// ---- GVLs/GlobalSettings.TcGVL
{attribute 'qualified_only'}
VAR_GLOBAL CONSTANT
	MAX_COMPONENTS: INT := 30;
	MAX_ALARMS: INT := 40;
END_VAR
{attribute 'qualified_only'}
VAR_GLOBAL PERSISTENT
	_dl:BOOL;
	{attribute 'TcEncoding':='UTF-8'}
	WebAdsAccessRoot: STRING := 'Main.GreenMaster';
	{attribute 'TcEncoding':='UTF-8'}
	PlcType: STRING := 'CX8190';
	PlcVersion: string := '1.0.33P5';
	Webname: STRING := 'NIBE AirSite GreenMaster';
	Users: ARRAY [0..24] OF User := [
		(Email := 'user', Password := 'user', Name := 'User', Permissions := Permissions.User),
		(Email := 'admin', Password := 'admin', Name := 'Admin', Permissions := Permissions.AdminUser),
		(Email := 'super', Password := 'super', Name := 'Super', Permissions := Permissions.SuperUser)
	];
	{attribute 'TcEncoding':='UTF-8'}
	SiteNames: ARRAY [0..99] OF STRING;
	Components: ARRAY [0..MAX_COMPONENTS - 1] OF Component := [
		(Name := ComponentNames.GM, EN := FALSE, Path := 'Main.GreenMaster', Required := TRUE, Permissions := Permissions.User),
		(Name := ComponentNames.GM_BASE, EN := TRUE, Path := 'Main.GreenMaster.Parameters', Required := TRUE, Resource := 'Parameter', Permissions := Permissions.User),
		(Name := ComponentNames.GM_IO, EN := TRUE, Path := 'Globals.IO', Required := TRUE, Resource := 'Parameter', Permissions := Permissions.User),
		(Name := ComponentNames.GM_VENT, EN := TRUE, Path := 'Main.GreenMaster.ParametersVENT', Resource := 'Parameter', Permissions := Permissions.User),
		(Name := ComponentNames.GM_XXL, EN := TRUE, Path := 'Main.GreenMaster.ParametersXXL', Resource := 'Parameter', Permissions := Permissions.User),
		(Name := ComponentNames.GM_A, EN := FALSE, Path := 'Main.GreenMaster.ParametersGMA', Resource := 'Parameter', Permissions := Permissions.User),
		(Name := ComponentNames.GM_C_F, EN := FALSE, Path := 'Main.GreenMaster.ParametersGMCF', Resource := 'Parameter', Permissions := Permissions.User),
		(Name := ComponentNames.GM_C_T, EN := FALSE, Path := 'Main.GreenMaster.ParametersGMCT', Resource := 'Parameter', Permissions := Permissions.User),
		(Name := ComponentNames.GM_SMOKE_CONTROL, EN := TRUE, Path := 'Main.GreenMaster.ParametersSC', Resource := 'Parameter', Permissions := Permissions.User),
		(Name := ComponentNames.SMOKE_CONTROL_ADS, EN := TRUE, Path := 'ADS_SmokeControl.Tags', Resource := 'Parameter', Permissions := Permissions.User),
		(Name := ComponentNames.GM_OPT_STD, EN := TRUE, Path := 'ADS_Standard.Tags', Resource := 'Parameter', Permissions := Permissions.User),
		(Name := ComponentNames.SIMULATION, EN := FALSE, Path := 'Main.GreenMaster.Simulation', Resource := 'Parameter', Permissions := Permissions.User),
		(Name := ComponentNames.REDUNDANCY, EN := FALSE, Path := 'Main.GreenMaster.Redundancy', Resource := 'Parameter', Permissions := Permissions.User),
		(Name := ComponentNames.EXTRA_ALARMS, EN := TRUE, Path := 'ADS_ExtraAlarms.Tags', Resource := 'Parameter', Permissions := Permissions.User),
		(Name := ComponentNames.PARALLEL_UNITS, EN := FALSE, Path := 'ADS_ParallelUnits.Tags', Resource := 'Parameter', Permissions := Permissions.User),
		(Name := ComponentNames.None)
	];
	AlarmDefs: ARRAY [0..MAX_ALARMS - 1] OF AlarmDef := [
		(Name := 'FireExtract', Polarity := AlarmPolarity.ActiveLow),
		(Name := '')
	];
END_VAR

// ---- POUs/Main.TcPOU
PROGRAM Main
VAR
	// JaWa
	_iDbg:INT;	
	_download5:BOOL;
	//Enum1: FanControlTypes := FanControlTypes.Flow;
	GreenMaster: GreenMasterXXL_FB;
	StartupDone: BOOL;
	EventLog: EventLog;
	xxx: bool;
	Saver: FB_S_UPS_CX81xx;
	HostName: FB_GetHostName;
	UseReverse_C_QN1: BOOL;
	test1: bool;
	
	Std_Interface : Standard_Interface;
	ExtraAlarms_Interface: ExtraAlarms_Interface;
	SmokeControl_Interface: SmokeControl_Interface;

	Redundancy:Redundancy;
	//ParallelUnits: ParallelUnits;
	
	GreenMasterDI: GreenMasterDI;
	GreenMasterDO: GreenMasterDO;
	GreenMasterAI: GreenMasterAI;
	GreenMasterAO: GreenMasterAO;
	GreenMasterAI2_RTU: GreenMasterAIU_ModbusRTU;
	AnySensorError: BOOL;
	{attribute 'TcEncoding':='UTF-8'}
	str: STRING;
	n: INT;
	
	DebugStop: BOOL;
	WritePersistentData: WritePersistentData;
	StartWritePersistentData: BOOL;
	SavedParameters: GreenMasterBaseParameters;
	DevMon: DeviationMonitor;
	DevValue: LREAL;
	TestPID: TestPID;
	fbTime : FB_LocalSystemTime := ( bEnable := TRUE, dwCycle := 1 );
	LastSecondsCounter: LINT;
    sTime: STRING;	
	sPart1: STRING;
	sPart2: STRING;
	ExceptionYet: BOOL;
	PTest: POINTER TO BYTE;
	Crash: BOOL;
	i: INT;
	w: WORD;
	Rr: LREAL;
	UseKL3464: BOOL;
	FreezeHysteresis: Hysteresis;
	CurrentFreezeAlarm: BOOL;
END_VAR
VAR PERSISTENT
END_VAR

IF NOT ExceptionYet THEN
	//__TRY
		EventLog(EventLogData := Globals.EventLog);
		IF NOT StartupDone THEN
			Globals.SystemStartTime := NowDT();
			EventLog.LogEvent(Message := 'Starting up', Kind := EventTypes.Information);
			//EventLog.LogEventJSON(Message := 'Test data $${KFactor} and $${PressureControl.SP}', Kind := EventTypes.Debug, VarAdr := ADR(GreenMaster.Parameters.Regulation.ExtractAir), VarSize := SIZEOF(GreenMaster.Parameters.Regulation.ExtractAir), VarType := 'AirParameters');
			Rr := 4;	
			i := -4;
			StartupDone := TRUE;
		END_IF
		SavedParameters := GreenMaster.GetParameters();
		Globals.SystemUpTime := DT_TO_DWORD(NowDT()) - DT_TO_DWORD(Globals.SystemStartTime);
		
		TestPID();
		
		str := '';
		FOR n := 0 TO GlobalSettings.MAX_COMPONENTS DO
			IF GlobalSettings.Components[n].Name = ComponentNames.NONE THEN
				EXIT;
			END_IF
			IF GlobalSettings.Components[n].EN THEN
				IF str <> '' THEN
					str := concat(str, ', ');
				END_IF
				str := concat(str, TO_STRING(GlobalSettings.Components[n].Name));
			END_IF
		END_FOR
		Globals.Components := str;
		
		HostName(bExecute := TRUE);
		// CX-503E98 CTH 1
		// CX-492F8F Diginet lab
		// CX-4F1CE6 NIBE AirSite lab
		// 
		Globals.HostName := HostName.sHostName; 
		IF F_ToUCase(HostName.sHostName) = 'CX-503E98' THEN
			UseReverse_C_QN1 := FALSE;
		ELSE
			UseReverse_C_QN1 := GreenMaster.Parameters.Io.AOutCalibration.C_QN1.InvertedOutput;
		END_IF
		
		IF F_ToUCase(HostName.sHostName) = 'STU_E6-LB02' THEN
			UseKL3464 := TRUE;
		END_IF
		IF (HostName.sHostName <> '') and (NOT GreenMaster.Parameters.System.ProjectDefaultSet) THEN			
			IF F_ToUCase(HostName.sHostName) = 'STU_E1-LB01' OR F_ToUCase(HostName.sHostName) = 'STU_E1-LB02' THEN
				GetComponent(Name := ComponentNames.PARALLEL_UNITS).EN := TRUE;
				GreenMaster.GetParameters().Regulation.Temperature.HeaterOutputDirection := HeaterOutputDirections.IncreaseToHeat;
				GreenMaster.GetParameters().Regulation.ExtractAir.Control.I := T#10M;
				GreenMaster.GetParameters().Regulation.SupplyAir.Control.I := T#10M;
				ADS_Standard.Tags.Settings.ExtractFanControl_I := GreenMaster.GetParameters().Regulation.ExtractAir.Control.I;
				ADS_Standard.Tags.Settings.SupplyFanControl_I := GreenMaster.GetParameters().Regulation.SupplyAir.Control.I;
				GreenMaster.GetParameters().Regulation.ExtractAir.KFactor := 151.4;
				GreenMaster.GetParameters().Regulation.ExtractAir.FireExhaust.EN := TRUE;
				GreenMaster.GetParameters().Regulation.ExtractAir.FireExhaust.Speed := 0.4;
				GreenMaster.GetParameters().Regulation.ExtractAir.FireSupply.EN := TRUE;
				GreenMaster.GetParameters().Regulation.ExtractAir.FireSupply.Speed := 0.4;
				GreenMaster.GetParameters().Regulation.SupplyAir.KFactor := 151.4;
				GreenMaster.GetParameters().Regulation.SupplyAir.FireExhaust.EN := FALSE;
				GreenMaster.GetParameters().Regulation.SupplyAir.FireExhaust.Speed := 0;
				GreenMaster.GetParameters().Alarm.Polarity.B.Tx1Fail := TRUE;
				GreenMaster.GetParameters().Alarm.Enabled.B.Pump1 := FALSE;
				ADS_ParallelUnits.Tags.Settings.SupplyAirSetPointAdjustment.Curve.Y1 := 160;
				ADS_ParallelUnits.Tags.Settings.SupplyAirSetPointAdjustment.Curve.Y2 := 160;
				ADS_ParallelUnits.Tags.Settings.SupplyAirSetPointAdjustment.Curve.Y3 := 160;
				ADS_ParallelUnits.Tags.Settings.SupplyAirSetPointAdjustment.Curve.Y4 := 160;
				ADS_ParallelUnits.Tags.Settings.SupplyAirSetPointAdjustment.Curve.Y5 := 160;
				ADS_ParallelUnits.Tags.Settings.SupplyAirSetPointAdjustment.Curve.Y6 := 160;
				ADS_ParallelUnits.Tags.Settings.SupplyAirSetPointAdjustment.Curve.Y7 := 160;
				ADS_ParallelUnits.Tags.Settings.SupplyAirSetPointAdjustment.Curve.Y8 := 160;
				ADS_ParallelUnits.Tags.Settings.SupplyAirSetPointAdjustment.Curve.Y9 := 160;
				
				ADS_ParallelUnits.Tags.Settings.ExtractAirSetPointAdjustment.Curve.Y1 := 150;
				ADS_ParallelUnits.Tags.Settings.ExtractAirSetPointAdjustment.Curve.Y2 := 150;
				ADS_ParallelUnits.Tags.Settings.ExtractAirSetPointAdjustment.Curve.Y3 := 150;
				ADS_ParallelUnits.Tags.Settings.ExtractAirSetPointAdjustment.Curve.Y4 := 150;
				ADS_ParallelUnits.Tags.Settings.ExtractAirSetPointAdjustment.Curve.Y5 := 150;
				ADS_ParallelUnits.Tags.Settings.ExtractAirSetPointAdjustment.Curve.Y6 := 150;
				ADS_ParallelUnits.Tags.Settings.ExtractAirSetPointAdjustment.Curve.Y7 := 150;
				ADS_ParallelUnits.Tags.Settings.ExtractAirSetPointAdjustment.Curve.Y8 := 150;
				ADS_ParallelUnits.Tags.Settings.ExtractAirSetPointAdjustment.Curve.Y9 := 150;
			END_IF
			IF F_ToUCase(HostName.sHostName) = 'STU_E6-LB03' THEN
				GreenMaster.GetParameters().Regulation.Temperature.HeaterOutputDirection := HeaterOutputDirections.DecreaseToHeat;
				GreenMaster.GetParameters().Regulation.ExtractAir.KFactor := 111;
				GreenMaster.GetParameters().Regulation.ExtractAir.FireExhaust.EN := FALSE;
				GreenMaster.GetParameters().Regulation.ExtractAir.FireExhaust.Speed := 0;
				GreenMaster.GetParameters().Regulation.ExtractAir.FireSupply.EN := FALSE;
				GreenMaster.GetParameters().Regulation.ExtractAir.FireSupply.Speed := 0;
				GreenMaster.GetParameters().Regulation.SupplyAir.KFactor := 111;
				GreenMaster.GetParameters().Regulation.SupplyAir.FireExhaust.EN := FALSE;
				GreenMaster.GetParameters().Regulation.SupplyAir.FireExhaust.Speed := 0;
				GreenMaster.GetParameters().Alarm.Polarity.B.Pump1 := TRUE;
			END_IF
			IF F_ToUCase(HostName.sHostName) = 'STU_E6-LB01' OR F_ToUCase(HostName.sHostName) = 'STU_E6-LB02' THEN
				GetComponent(Name := ComponentNames.PARALLEL_UNITS).EN := TRUE;
				GreenMaster.GetParameters().Regulation.Temperature.HeaterOutputDirection := HeaterOutputDirections.IncreaseToHeat;
				GreenMaster.GetParameters().Regulation.ExtractAir.KFactor := 111;
				GreenMaster.GetParameters().Regulation.ExtractAir.FireExhaust.EN := FALSE;
				GreenMaster.GetParameters().Regulation.ExtractAir.FireExhaust.Speed := 0;
				GreenMaster.GetParameters().Regulation.SupplyAir.KFactor := 111;
				GreenMaster.GetParameters().Regulation.SupplyAir.FireExhaust.EN := FALSE;
				GreenMaster.GetParameters().Regulation.SupplyAir.FireExhaust.Speed := 0;
				GreenMaster.GetParameters().Alarm.Polarity.B.Tx1Fail := TRUE;
			END_IF
			IF F_ToUCase(HostName.sHostName) = 'AIRPLC-DEMO' THEN
				GetComponent(Name := ComponentNames.PARALLEL_UNITS).EN := TRUE;
				GetComponent(Name := ComponentNames.SIMULATION).EN := TRUE;
				GreenMaster.GetParameters().System.Operation.Simulation := TRUE;
				GreenMaster.GetParameters().Regulation.Temperature.HeaterOutputDirection := HeaterOutputDirections.IncreaseToHeat;
				GreenMaster.GetParameters().Regulation.ExtractAir.KFactor := 111;
				GreenMaster.GetParameters().Regulation.ExtractAir.FireExhaust.EN := FALSE;
				GreenMaster.GetParameters().Regulation.ExtractAir.FireExhaust.Speed := 0;
				GreenMaster.GetParameters().Regulation.SupplyAir.KFactor := 111;
				GreenMaster.GetParameters().Regulation.SupplyAir.FireExhaust.EN := FALSE;
				GreenMaster.GetParameters().Regulation.SupplyAir.FireExhaust.Speed := 0;
				//GreenMaster.GetParameters().Regulation.SupplyAir.MaxSpeed := 0.4;
				//GreenMaster.GetParameters().Regulation.ExtractAir.MaxSpeed := 0.4;
			END_IF
			IF F_ToUCase(HostName.sHostName) = 'CX-662AA1' THEN
				GetComponent(Name := ComponentNames.PARALLEL_UNITS).EN := TRUE;
				GetComponent(Name := ComponentNames.SIMULATION).EN := TRUE;
				GreenMaster.GetParameters().System.Operation.Simulation := TRUE;
				GreenMaster.GetParameters().Regulation.Temperature.HeaterOutputDirection := HeaterOutputDirections.IncreaseToHeat;
				GreenMaster.GetParameters().Regulation.ExtractAir.KFactor := 111;
				GreenMaster.GetParameters().Regulation.ExtractAir.FireExhaust.EN := FALSE;
				GreenMaster.GetParameters().Regulation.ExtractAir.FireExhaust.Speed := 0;
				GreenMaster.GetParameters().Regulation.SupplyAir.KFactor := 111;
				GreenMaster.GetParameters().Regulation.SupplyAir.FireExhaust.EN := FALSE;
				GreenMaster.GetParameters().Regulation.SupplyAir.FireExhaust.Speed := 0;
				GreenMaster.GetParameters().Regulation.SupplyAir.MaxSpeed := 0.4;
				GreenMaster.GetParameters().Regulation.ExtractAir.MaxSpeed := 0.4;
			END_IF
			IF (F_ToUCase(HostName.sHostName) = 'DIGINET-1') or (F_ToUCase(HostName.sHostName) = 'DIGINET-2') THEN
				GetComponent(Name := ComponentNames.PARALLEL_UNITS).EN := TRUE;
				GetComponent(Name := ComponentNames.SIMULATION).EN := TRUE;
				GreenMaster.GetParameters().System.Operation.Simulation := TRUE;
				GreenMaster.GetParameters().Regulation.Temperature.HeaterOutputDirection := HeaterOutputDirections.IncreaseToHeat;
				GreenMaster.GetParameters().Regulation.ExtractAir.KFactor := 111;
				GreenMaster.GetParameters().Regulation.ExtractAir.FireExhaust.EN := TRUE;
				GreenMaster.GetParameters().Regulation.ExtractAir.FireExhaust.Speed := 0.5;
				GreenMaster.GetParameters().Regulation.SupplyAir.KFactor := 111;
				GreenMaster.GetParameters().Regulation.SupplyAir.FireExhaust.EN := FALSE;
				GreenMaster.GetParameters().Regulation.SupplyAir.FireExhaust.Speed := 0;
				GreenMaster.GetParameters().system.Operation.StartupHeatRecoveryTime := T#30S;
				GreenMaster.GetParameters().system.Operation.ExhaustFanStartupDelay := T#10S;
				GreenMaster.GetParameters().system.Operation.SupplyFanStartupDelay := T#20S;
				GreenMaster.GetParameters().system.Operation.StartupDamperWaitTime := T#5S;
			END_IF
			GreenMaster.GetParameters().System.ProjectDefaultSet := TRUE;
		END_IF
		
		IF GreenMaster.Parameters.System.Operation.IoUpdateEN THEN
			GreenMasterDI(DIn := Globals.IO.DIn, DInLevels := GreenMaster.Parameters.IO.DInLevels);
			GreenMasterDO(DOut := Globals.IO.DOut);
			GreenMasterAI(AIn := Globals.IO.AIn);
			GreenMasterAO(AOut := Globals.IO.AOut);
			GreenMasterAI2_RTU(Parameters:=GreenMaster.GetParameters(), EN:= TRUE);
		END_IF
		
		Std_Interface(EN := GetComponent(Name := ComponentNames.GM_OPT_STD).EN, AIn := Globals.IO.AIn);
		
		// Redundant drift
		IF GetComponent(Name := ComponentNames.REDUNDANCY).EN THEN
			Redundancy(	EN := GetComponent(Name := ComponentNames.REDUNDANCY).EN,
						_UPPSTART_DONE:=StartupDone,
						_TF_CMD:=GreenMaster.Parameters.Regulation.SupplyAir.Control.CV > 0,
						_TF_V:=GreenMaster.Parameters.Regulation.SupplyAir.Control.CV > 0 AND GreenMaster.GetCurrentSupplyAirPV() > 10,
						_TF_OP:=LREAL_TO_REAL(GreenMaster.Parameters.Regulation.SupplyAir.Control.CV),
						_TL_GP_PV:=LREAL_TO_REAL(GreenMaster.GetCurrentSupplyAirPV()),
						_FF_CMD:=GreenMaster.Parameters.Regulation.ExtractAir.Control.CV > 0,
						_FF_V:=GreenMaster.Parameters.Regulation.ExtractAir.Control.CV > 0 AND GreenMaster.GetCurrentExtractAirPV() > 10,
						_FF_OP:=LREAL_TO_REAL(GreenMaster.Parameters.Regulation.ExtractAir.Control.CV),
						_FL_GP_PV:=LREAL_TO_REAL(GreenMaster.GetCurrentExtractAirPV()),
						_SERVICEBRYTARE:=FALSE
						);
		END_IF
		// Parallel units
		(*
		IF GetComponent(Name := ComponentNames.PARALLEL_UNITS).EN THEN
			ParallelUnits(	EN := GetComponent(Name := ComponentNames.PARALLEL_UNITS).EN,
							Tags := ADS_ParallelUnits.Tags,
							Parameters := GreenMaster.Parameters 
						);
		END_IF
		*)
		IF GetComponent(Name := ComponentNames.GM_BASE).EN THEN
			GreenMaster.Update(DO_ := GreenMasterDO, AO := GreenMasterAO);
			GreenMaster(
				EN := TRUE AND (NOT DebugStop),
				RemoteEN := GreenMaster.Parameters.System.Operation.RemoteEN, //Std_Interface.ENO OR CTH_Interface.ENO OR Stena_Interface.ENO,	// TODO: Varför bara CTH här i original?  
				DI := GreenMasterDI,
				AI := GreenMasterAI,
				AI2 := GreenMasterAI2_RTU,
				TCP_AI := SmokeControl.GreenMasterSmokeControl,  
				Reverse_C_QN1 := UseReverse_C_QN1,
				NightCooling := GreenMaster.Parameters.Regulation.NightCooling,
				EnableFansAndDampers := Std_Interface.EN,
				ExtraFireSupplyAlarm := FALSE, //ParallelUnits.FireSupplyAlarm,
				ExtraFireExtractAlarm := FALSE //ParallelUnits.FireExtractAlarm
			);
		END_IF
		
		IF GetComponent(Name := ComponentNames.SIMULATION).EN THEN
			IF GreenMaster.GetParameters().System.Operation.Simulation THEN
				GreenMaster.Simulation(Parameters := GreenMaster.GetParameters(), Simulation := GreenMaster.GetParameters().Simulation);			
			END_IF
		END_IF
		
		AnySensorError := GreenMaster.Parameters.IO.AIn.F_BT1_Error OR 
			GreenMaster.Parameters.IO.AIn.T_BT2_Error OR
			GreenMaster.Parameters.IO.AIn.T_BT3_Error OR
			GreenMaster.Parameters.IO.AIn.H_BT1_Error OR
			GreenMaster.Parameters.IO.AIn.T_BT1_Error OR
			GreenMaster.Parameters.IO.AIn.BT1_Error OR
			GreenMaster.Parameters.IO.AIn.BT2_Error OR
			GreenMaster.Parameters.IO.AIn.F_BT2_Error OR	
			GreenMaster.Parameters.IO.AIn.F_BP1_Error OR
			GreenMaster.Parameters.IO.AIn.T_BP1_Error OR
			GreenMaster.Parameters.IO.AIn.F_BP2_Error OR
			GreenMaster.Parameters.IO.AIn.T_BP2_Error OR
			GreenMaster.Parameters.IO.AIn.F_BP3_Error OR
			GreenMaster.Parameters.IO.AIn.T_BF1_Error OR
			GreenMaster.Parameters.IO.AIn.F_BF1_Error;	
		
		
		// Save persistent data on power off or fail
		Saver();
		WritePersistentData(NETID := '', PORT := 851, TMOUT := T#10S, START := StartWritePersistentData);
		
		DevMon(Value := DevValue, TargetValue := 5);
		
		IF GetComponent(Name := ComponentNames.EXTRA_ALARMS).EN THEN	
			GreenMaster.GetParameters().Alarm.Status.A.AL01 := NOT ExtraAlarmInputs.AL01;
			GreenMaster.GetParameters().Alarm.Status.A.AL02 := NOT ExtraAlarmInputs.AL02;
			GreenMaster.GetParameters().Alarm.Status.A.AL03 := NOT ExtraAlarmInputs.AL03;
			GreenMaster.GetParameters().Alarm.Status.A.AL04 := NOT ExtraAlarmInputs.AL04;
			GreenMaster.GetParameters().Alarm.Status.A.AL05 := NOT ExtraAlarmInputs.AL05;
			GreenMaster.GetParameters().Alarm.Status.A.AL06 := NOT ExtraAlarmInputs.AL06;
			GreenMaster.GetParameters().Alarm.Status.A.AL07 := NOT ExtraAlarmInputs.AL07;
			GreenMaster.GetParameters().Alarm.Status.A.AL08 := NOT ExtraAlarmInputs.AL08;
		END_IF
		ExtraAlarms_Interface(EN := GetComponent(Name := ComponentNames.EXTRA_ALARMS).EN);
		SmokeControl_Interface(EN := GetComponent(Name := ComponentNames.GM_SMOKE_CONTROL).EN);
		fbtime();
		IF Globals.SecondsCounter <> LastSecondsCounter THEN
			LastSecondsCounter := Globals.SecondsCounter;
			// 2021-11-10-08:08:53.582
			sTime := SYSTEMTIME_TO_STRING(fbTime.systemTime);
			sPart1 := Delete(sTime, 4, 20);
			sPart2 := Replace(sPart1, ' ', 1, 11);
			GreenMaster.GetParameters().System.SystemTime := sPart2;
		END_IF
	//__CATCH
	//	ExceptionYet := TRUE; 			
	//__ENDTRY
ELSE
	ExceptionYet := TRUE; 	
END_IF

FreezeHysteresis(Value := GreenMaster.GetParameters().IO.AIn.H_BT1, LimitValue := GreenMaster.GetParameters().Alarm.Limits.A.Freeze, Offset := 0.5);
CurrentFreezeAlarm := FreezeHysteresis.Below OR GreenMaster.GetParameters().IO.AIn.H_BT1_Error;
GreenMaster.GetParameters().Alarm.Status.A.Freeze := CurrentFreezeAlarm  (*OR	ParallelUnits.FreezeAlarm*);

END_PROGRAM

// ---- POUs/GreenMasterXXL_FB.TcPOU
FUNCTION_BLOCK GreenMasterXXL_FB EXTENDS GreenMasterXXL
VAR_INPUT
END_VAR
VAR_OUTPUT
END_VAR
VAR
END_VAR


// PAGE Overview
Super^(); // GreenMasterXXL

END_FUNCTION_BLOCK

// ---- DUTs/GreenMaster/GreenMasterXXL.TcPOU
FUNCTION_BLOCK GreenMasterXXL EXTENDS GreenMasterBase
VAR
	ParametersXXLFB: GreenMasterParametersXXLFB;
END_VAR
VAR PERSISTENT
	ParametersXXL: GreenMasterParametersXXL;
END_VAR
VAR_INPUT
END_VAR
VAR_OUTPUT
END_VAR
VAR
	SupplyFanControl: FanControl;
	ExtractFanControl: FanControl;
	Recirculation: BOOL;
	VentilationControl: VentilationControl;
	ExhaustAir: BOOL;
	SupplyAir: BOOL := TRUE;
	StopVentilation: bool;

	ExtractFanPV: LREAL;
	SupplyFanPV: LREAL;
	Defrost_0: Defrost;
	WriteLRealIf_0: WriteLRealIf;
END_VAR
VAR // added by the converter: edge detectors and wires of the graphical bodies
    _w1, _w2, _w3, _w4 : ANY;
END_VAR


// PAGE Base functionality Inherited from greenMasterBase
Super^(); // GreenMasterBase

// PAGE Ventilation
Ventilation := VentilationControl.ENO;
VentilationControl(EN := Parameters.Regulation.Control.EN AND SystemStateVentilation AND ENO AND NOT StopVentilation);
VentilationRunning := VentilationControl.ENO;

// PAGE Supply Air
Parameters.Regulation.SupplyAir.Control.CV := SupplyFanControl.CV;
_w1 := Parameters.Alarm.Active.B.SupplyFan OR Parameters.Alarm.Active.B.ExtractFan;
WriteLRealIf_0(Out := Parameters.IO.AOut.T_GQ1, EN := TRUE, In := SupplyFanControl.CV); // WriteLRealIf
// Output via VAR_IN_OUT
SupplyFanControl(
    Parameters := Parameters,
    EN := Ventilation,
    ControlMode := Parameters.Regulation.SupplyAir.ControlMode,
    ControlParameters := Parameters.Regulation.SupplyAir.Control,
    Pressure := Parameters.IO.AIn.T_BP1,
    PressureError := Parameters.IO.Status.SensorStatus.T_BP1 <> 'OK',
    Flow := Parameters.IO.AIn.T_BF1,
    FlowError := Parameters.IO.Status.SensorStatus.T_BF1 <> 'OK',
    MasterPV := ExtractFanPV,
    FanAlarm := _w1,
    MinSpeed := Parameters.Regulation.SupplyAir.MinSpeed,
    MaxSpeed := Parameters.Regulation.SupplyAir.MaxSpeed,
    ExtendedOperation := _w2,
    PostVentilationTime := Parameters.System.Operation.PostVentilationTime,
    FireExhaust := GetFireExtractAlarms(),
    Damper := Parameters.IO.DOut.T_QM2,
    FireExhaustPar := Parameters.Regulation.SupplyAir.FireExhaust,
    FireSupplyPar := Parameters.Regulation.SupplyAir.FireSupply,
    FireSupply := Parameters.Alarm.Active.A.FireSupply); // FanControl
SupplyFanPV := SupplyFanControl.PV;
Parameters.IO.DOut.T_RUN := SupplyFanControl.FanRunning;
Parameters.IO.DOut.R_QM1 := SupplyFanControl.Recirculation;
_w2 := NightCooling OR DI.ExtendedOperation OR Parameters.System.Operation.TimeChannels.HighSpeed;

// PAGE Extract Air
_w3 := NightCooling OR DI.ExtendedOperation OR Parameters.System.Operation.TimeChannels.HighSpeed;
Parameters.Regulation.ExtractAir.Control.CV := ExtractFanControl.CV;
_w4 := Parameters.Alarm.Active.B.SupplyFan OR Parameters.Alarm.Active.B.ExtractFan;
WriteLRealIf_0(Out := Parameters.IO.AOut.F_GQ1, EN := TRUE, In := ExtractFanControl.CV); // WriteLRealIf
// Output via VAR_IN_OUT
ExtractFanControl(
    Parameters := Parameters,
    EN := Ventilation,
    ControlMode := Parameters.Regulation.ExtractAir.ControlMode,
    ControlParameters := Parameters.Regulation.ExtractAir.Control,
    Pressure := Parameters.IO.AIn.F_BP1,
    PressureError := Parameters.IO.Status.SensorStatus.F_BP1 <> 'OK',
    Flow := Parameters.IO.AIn.F_BF1,
    FlowError := Parameters.IO.Status.SensorStatus.F_BF1 <> 'OK',
    MasterPV := SupplyFanPV,
    FanAlarm := _w4,
    MinSpeed := Parameters.Regulation.ExtractAir.MinSpeed,
    MaxSpeed := Parameters.Regulation.ExtractAir.MaxSpeed,
    ExtendedOperation := _w3,
    PostVentilationTime := Parameters.System.Operation.PostVentilationTime,
    FireExhaust := GetFireExtractAlarms(),
    Damper := Parameters.IO.DOut.F_QM1,
    FireExhaustPar := Parameters.Regulation.ExtractAir.FireExhaust,
    FireSupplyPar := Parameters.Regulation.ExtractAir.FireSupply,
    FireSupply := Parameters.Alarm.Active.A.FireSupply); // FanControl
ExtractFanPV := ExtractFanControl.PV;
Parameters.IO.DOut.F_RUN := ExtractFanControl.FanRunning;

// PAGE Defrost
Defrost_0(
    Parameters := Parameters,
    EN := Parameters.System.Defrost.EN AND NOT Parameters.Alarm.Active.A.FireSupply AND NOT (GetFireExtractAlarms()),
    Temperature := Parameters.IO.AIn.T_BT2,
    Pressure := Parameters.IO.AIn.F_BP3); // Defrost

METHOD ExtractFanOverride : BOOL
VAR_INPUT
	Override: BOOL;
	Speed: LREAL;
END_VAR
VAR_INST
	LastExtractOverrideCV: lreal;
END_VAR
ExtractFanControl.Override := Override;
ExtractFanControl.OverrideCV := Speed;
ExtractFanControl.SyncCV := LastExtractOverrideCV;
IF Speed > 0 THEN
	LastExtractOverrideCV := Speed;
END_IF
END_METHOD

METHOD Fire : BOOL
VAR_INPUT
END_VAR
SUPER^.Fire();
SupplyFanControl.Override := Parameters.Regulation.SupplyAir.FireExhaust.EN;
SupplyFanControl.OverrideCV := Parameters.Regulation.SupplyAir.FireExhaust.Speed;
ExtractFanControl.Override := Parameters.Regulation.ExtractAir.FireExhaust.EN;
ExtractFanControl.OverrideCV := Parameters.Regulation.ExtractAir.FireExhaust.Speed;
END_METHOD

METHOD FireEnd : BOOL
VAR_INPUT
END_VAR
SUPER^.FireEnd();
SupplyFanControl.Override := FALSE;
SupplyFanControl.OverrideCV := 0;
ExtractFanControl.Override := FALSE;
ExtractFanControl.OverrideCV := 0;
END_METHOD

METHOD FireSupply : BOOL
VAR_INPUT
END_VAR
SUPER^.FireSupply();
CloseDampers();
StopVentilation := TRUE;
END_METHOD

METHOD FireSupplyEnd : BOOL
VAR_INPUT
END_VAR
SUPER^.FireSupplyEnd();
StopVentilation := FALSE;
END_METHOD

METHOD GetParametersXXL : REFERENCE TO GreenMasterParametersXXL
VAR_INPUT
END_VAR
GetParametersXXL := ParametersXXL;
END_METHOD

{attribute 'TcRpcEnable'}
METHOD Sum : LREAL
VAR_INPUT
	v1: LREAL;
	v2: LREAL;
END_VAR
Sum := v1 + v2;
END_METHOD

METHOD SupplyFanOverride : BOOL
VAR_INPUT
	Override: BOOL;
	Speed: LREAL;
END_VAR
VAR_INST
	LastSupplyOverrideCV: lreal;
END_VAR
SupplyFanControl.Override := Override;
SupplyFanControl.OverrideCV := Speed;
SupplyFanControl.SyncCV := LastSupplyOverrideCV;
IF Speed > 0 THEN
	LastSupplyOverrideCV := Speed;
END_IF
END_METHOD

METHOD Update : BOOL
VAR_INPUT
	DO_: REFERENCE TO GreenMasterDO_Base;
	AO: REFERENCE TO GreenMasterAO_Base;
END_VAR
SUPER^.Update(DO_, AO);
IF Parameters.System.Operation.EN THEN
	SupplyAir := NOT Recirculation;	
END_IF
END_METHOD

END_FUNCTION_BLOCK

// ---- DUTs/GreenMaster/GreenMasterBase.TcPOU
FUNCTION_BLOCK GreenMasterBase
VAR
	ParametersFB: GreenMasterBaseParametersFB;
	ParametersSCFB: SmokeControlParametersBaseFB;
	Hysteresis_5: Hysteresis;
	Hysteresis_6: Hysteresis;
	T_BT2_BelowCoolingLimit: BOOL;
	SupplyIf: WriteBoolIf;
	ExerciseF_P1_0: ExerciseF_P1;
	SupplyDevMonParallell: DeviationMonitor;
	ExtractDevMonParallell: DeviationMonitor;
END_VAR
VAR PERSISTENT
	Parameters: GreenMasterBaseParameters;
	ParametersSC: SmokeControlParametersBase;
	Simulation: SimulationFB;
END_VAR
VAR_INPUT
	EN: BOOL := TRUE;
	RemoteEN: BOOL;
	DI: GreenMasterDI_Base;
	AI: GreenMasterAI_Base;
	AI2: GreenMasterAIU_Base;
	TCP_AI: GreenMasterSmokeControl_Base;
	Reverse_C_QN1: BOOL := TRUE;
	NightCooling: BOOL;
	EnableFansAndDampers: BOOL := TRUE;
	ExtraFireSupplyAlarm: BOOL := FALSE;
	ExtraFireExtractAlarm: BOOL := FALSE;
END_VAR
VAR_OUTPUT
	ENO: BOOL;
	VentilationRunning: BOOL;
	TemperatureControlRunning: BOOL;
	ExerciseF_QM2: ExerciseF_QM2;
END_VAR
VAR
	StateStartTime: LTIME;
	Ventilation: BOOL;
	SystemStateVentilation: BOOL;
	AlarmMonitor: AlarmMonitor;
	Hysteresis_0: Hysteresis;
	Hysteresis_1: Hysteresis;
	
	Scale1: Scale;
	Scale2: Scale;
	Scale3: Scale;
	TemperatureController: PidController;
	TP1: TP;
	TON1: TON;
	C_QN1_Low: LREAL;
	C_QN1_High: LREAL;
	
	test: BOOL;
	Av: Average;
	Pump1_TON: TON;
	Pump2_TON: TON;
	FreezeControl: BOOL;
	FreezeControlENO: BOOL;
	TempCV: LREAL;
	FreezeControlCV: LREAL;
	FreezeController: PidController;
	Hysteresis_2: Hysteresis;
	Hysteresis_3: Hysteresis;
	Hysteresis_4: Hysteresis;
	FireAlarmExtractAirTemperatureHysteresis: Hysteresis;
	FireAlarmExtractAirPressureTemperatureHysteresis: Hysteresis;
	FireAlarmExtractAirPressureHysteresis: Hysteresis;
	WriteLRealOnlyIf_0: WriteLRealOnlyIf;
	ColdRecyclingHysteresis: Hysteresis;
	TempDevMon: DeviationMonitor;
	SupplyDevMon: DeviationMonitor;
	ExtractDevMon: DeviationMonitor;
END_VAR
VAR // added by the converter: edge detectors and wires of the graphical bodies
    _w1, _w2, _w3, _w5 : BOOL;
    _w4, _w6, _w7, _w8 : ANY;
END_VAR


// PAGE System
ENO := (EN AND Parameters.System.Operation.EN AND (NOT Parameters.Alarm.Active.A.Fuse) AND (Parameters.IO.DIn.AUTO XOR Parameters.IO.DIn.HAND)) AND TRUE;

// PAGE Alarms
Parameters.Alarm.Status.B.RegulationDeviation := TempDevMon.Error;
Pump2_TON(IN := Globals.IO.DOut.DO16 XOR Globals.IO.DIn.DI22, PT := Parameters.Alarm.Delay.B.Pump2); // TON
_w1 := TRUE AND Pump2_TON.Q;
SupplyIf(
    Out := Parameters.Alarm.Status.B.ExtractAirDeviation,
    EN := Parameters.Regulation.SupplyAir.ControlMode <> FanControlTypes.Const,
    In := ExtractDevMon.Error); // WriteBoolIf
Parameters.Alarm.Status.B.Pump2 := _w1;
Parameters.Alarm.Status.B.SupplyFilter := Hysteresis_3.Above;
Parameters.Alarm.Status.A.FireSupply := Parameters.IO.DIn.FireSupplyAlarm OR ExtraFireSupplyAlarm;
Hysteresis_3(
    Value := Parameters.IO.AIn.T_BP2,
    LimitValue := Parameters.Alarm.Limits.B.SupplyFilter,
    Offset := 5); // Hysteresis
AlarmMonitor(
    AlarmLog := Globals.AlarmLog,
    EN := EN,
    Reset := Parameters.Alarm.Control.ResetAlarms,
    Parameters := Parameters);
Parameters.IO.DOut.AL_A := AlarmMonitor.AlarmA;
Parameters.IO.DOut.AL_B := AlarmMonitor.AlarmB;
Parameters.IO.DOut.AL_C := AlarmMonitor.AlarmC;
Parameters.IO.DOut.AL_D := AlarmMonitor.AlarmD;
Parameters.Alarm.Status.B.SmokeDetectorServiceExtract := Parameters.IO.DIn.ServiceAlarmCentralAndSmokeExhaustAir;
Parameters.Alarm.Status.B.ExtractFilter := Hysteresis_4.Above;
_w2 := Parameters.IO.DIn.FireExtractAlarm OR ExtraFireExtractAlarm;
Parameters.Alarm.Status.B.DamperError := SmokeControl.GreenMasterSmokeControl.DamperError;
Parameters.Alarm.Status.B.SmokeDetectorServiceSupply := Parameters.IO.DIn.ServiceAlarmSupplyAir;
Parameters.Alarm.Status.B.DamperModuleService := SmokeControl.GreenMasterSmokeControl.ServiceAlarm;
Parameters.Alarm.Status.C.SensorFailure := Main.AnySensorError;
Parameters.Alarm.Status.B.ExtractFan := Parameters.IO.DIn.F_GQ1_Alarm;
Hysteresis_4(
    Value := Parameters.IO.AIn.F_BP2,
    LimitValue := Parameters.Alarm.Limits.B.ExtractFilter,
    Offset := 5); // Hysteresis
Parameters.Alarm.Status.A.Fuse := Parameters.IO.DIn.FuseAlarm;
SupplyDevMon(
    EN := Parameters.Regulation.SupplyAir.ControlMode <> FanControlTypes.Const,
    Value := Parameters.Regulation.SupplyAir.Control.PV,
    TargetValue := Parameters.Regulation.SupplyAir.Control.CSP,
    DiffAllowed := Parameters.Alarm.Limits.B.SupplyAirPressureDeviation,
    Mode := DeviationMonitorMode.Diff,
    OnDelay := TIME_TO_LTIME(Parameters.Alarm.Delay.B.SupplyAirDeviation)); // DeviationMonitor
_w3 := TRUE AND Pump1_TON.Q;
Pump1_TON(IN := Parameters.IO.DOut.H_GP1 XOR Parameters.IO.DIn.H_GP1_Running, PT := Parameters.Alarm.Delay.B.Pump1); // TON
SupplyIf(
    Out := Parameters.Alarm.Status.B.SupplyAirDeviation,
    EN := Parameters.Regulation.SupplyAir.ControlMode <> FanControlTypes.Const,
    In := SupplyDevMon.Error); // WriteBoolIf
Parameters.Alarm.Status.B.Pump1 := _w3;
Parameters.Alarm.Status.B.SupplyFan := Parameters.IO.DIn.T_GQ1_Alarm;
TempDevMon(
    Value := Parameters.Regulation.Temperature.Control.PV,
    TargetValue := Parameters.Regulation.Temperature.Control.CSP,
    DiffAllowed := Parameters.Alarm.Limits.B.RegulationDeviation,
    Mode := DeviationMonitorMode.Diff,
    OnDelay := TIME_TO_LTIME(Parameters.Alarm.Delay.B.RegulationDeviation)); // DeviationMonitor
ExtractDevMon(
    EN := Parameters.Regulation.SupplyAir.ControlMode <> FanControlTypes.Const,
    Value := Parameters.Regulation.ExtractAir.Control.PV,
    TargetValue := Parameters.Regulation.ExtractAir.Control.CSP,
    DiffAllowed := Parameters.Alarm.Limits.B.ExtractAirPressureDeviation,
    Mode := DeviationMonitorMode.Diff,
    OnDelay := TIME_TO_LTIME(Parameters.Alarm.Delay.B.ExtractAirDeviation)); // DeviationMonitor
Parameters.Alarm.Status.B.Tx1Fail := Parameters.IO.DIn.TX1_Running;
SupplyIf(Out := Parameters.Alarm.Status.B.SupplyAirDeviation, EN := false, In := SupplyDevMonParallell.Error); // WriteBoolIf
SupplyDevMonParallell(
    EN := false,
    Value := Parameters.IO.AIn.T_BP1,
    TargetValue := ADS_ParallelUnits.Tags.Status.PressureSupplyCSP,
    DiffAllowed := Parameters.Alarm.Limits.B.SupplyAirPressureDeviation,
    Mode := DeviationMonitorMode.Diff,
    OnDelay := TIME_TO_LTIME(Parameters.Alarm.Delay.B.SupplyAirDeviation)); // DeviationMonitor
SupplyIf(
    Out := Parameters.Alarm.Status.B.ExtractAirDeviation,
    EN := false,
    In := ExtractDevMonParallell.Error); // WriteBoolIf
ExtractDevMonParallell(
    EN := false,
    Value := Parameters.IO.AIn.F_BP1,
    TargetValue := ADS_ParallelUnits.Tags.Status.PressureExtractCSP,
    DiffAllowed := Parameters.Alarm.Limits.B.ExtractAirPressureDeviation,
    Mode := DeviationMonitorMode.Diff,
    OnDelay := TIME_TO_LTIME(Parameters.Alarm.Delay.B.ExtractAirDeviation)); // DeviationMonitor

// PAGE Temperature Control
_w4 := MAX(FreezeControlCV, Scale1.u);
WriteLRealOnlyIf_0(EN := VentilationRunning, In := Scale2.u, InNotEN := Parameters.IO.AOut.F_QN1); // WriteLRealOnlyIf
TempCV := TemperatureController.CV;
_w5 := Parameters.Regulation.Temperature.EN AND VentilationRunning AND ENO AND (NOT NightCooling);
Hysteresis_5(Value := Parameters.IO.AIn.T_BT2, LimitValue := 5, Offset := 0.5); // Hysteresis
_w6 := Hysteresis_5.Below OR Hysteresis_0.Above OR ExerciseF_P1_0.Exercising;
TemperatureControlRunning := _w5;
_w7 := Parameters.Regulation.Temperature.Control.I / 5;
_w8 := LREAL_BMUX(B := NOT (FireAlarm()) AND ColdRecyclingHysteresis.Below, F := WriteLRealOnlyIf_0.Out, T := ParametersFB.Regulation.Temperature.MinOutput());
TemperatureController(
    EN := _w5,
    SP := Parameters.Regulation.Temperature.Control.CSP,
    PV := GetCurrentPV(),
    SyncCV := 0.875,
    Sync := _w5,
    I := Parameters.Regulation.Temperature.Control.I,
    P := Parameters.Regulation.Temperature.Control.P,
    DampingTime := _w7); // PidController
Scale1(EN := TemperatureController.ENO, x := TemperatureController.CV, x1 := 0.75, x2 := 1, u1 := 0, u2 := 1); // Scale
Parameters.IO.AOut.H_QN1 := _w4;
Hysteresis_0(Value := _w4, LimitValue := 0.02, Offset := 0.01); // Hysteresis
Parameters.IO.DOut.H_GP1 := _w6;
Scale2(
    x := TempCV,
    x1 := 0.25,
    x2 := 0.75,
    u1 := ParametersFB.Regulation.Temperature.MinOutput(),
    u2 := ParametersFB.Regulation.Temperature.MaxOutput()); // Scale
Parameters.IO.AOut.F_QN1 := _w8;
Scale3(
    EN := TemperatureController.ENO AND NOT T_BT2_BelowCoolingLimit,
    x := TemperatureController.CV,
    x1 := 0,
    x2 := 0.25,
    u1 := C_QN1_Low,
    u2 := C_QN1_High); // Scale
Parameters.IO.AOut.C_QN1 := Scale3.u;
Hysteresis_1(
    EN := TemperatureController.ENO,
    Value := TemperatureController.CV,
    LimitValue := 0.25,
    Offset := 0.01); // Hysteresis
Parameters.IO.DOut.C_GP1 := Hysteresis_1.ENO AND Hysteresis_1.Below AND NOT Hysteresis_6.Below;
Hysteresis_6(Value := Parameters.IO.AIn.T_BT2, LimitValue := 12, Offset := 0.5); // Hysteresis
T_BT2_BelowCoolingLimit := Hysteresis_6.Below;

// PAGE Service Service, test, exercise
ExerciseF_QM2(Parameters := Parameters);
ExerciseF_P1_0(Parameters := Parameters); // ExerciseF_P1

// PAGE Freeze Control
FreezeController(
    EN := Hysteresis_2.Below,
    SP := Parameters.Regulation.Temperature.FreezeGuardControl.SP,
    PV := Parameters.IO.AIn.H_BT1,
    P := Parameters.Regulation.Temperature.FreezeGuardControl.P,
    I := Parameters.Regulation.Temperature.FreezeGuardControl.I); // PidController
FreezeControl := Hysteresis_2.Below;
Hysteresis_2(
    Value := Parameters.IO.AIn.H_BT1,
    LimitValue := Parameters.Regulation.Temperature.FreezeGuardLimit,
    Offset := Parameters.Regulation.Temperature.FreezeGuardHysteresis); // Hysteresis
FreezeControlENO := FreezeController.ENO;
FreezeControlCV := FreezeController.CV;

// PAGE Alarms
Parameters.Alarm.Status.A.FireExtract := _w2;
// Parameters.System.Operation.RemoteEN: input not connected
// not FreezeControl: input not connected

METHOD CloseDampers : BOOL
VAR_INPUT
END_VAR
Parameters.IO.DOut.T_QM2 := FALSE;
Parameters.IO.DOut.F_QM1 := FALSE;
Parameters.IO.DOut.F_QM2 := TRUE;
Parameters.IO.DOut.R_QM1 := FALSE;
Parameters.IO.DOut.T_QM1_1 := FALSE;
Parameters.IO.DOut.T_QM1_2 := FALSE;
Parameters.IO.DOut.T_QM1_3 := FALSE;
Parameters.IO.DOut.T_QM1_4 := FALSE;
Parameters.IO.DOut.T_QM1_5 := FALSE;
Parameters.IO.DOut.T_QM1_6 := FALSE;
END_METHOD

METHOD DampersOpen : BOOL
VAR_INPUT
END_VAR
DampersOpen := ParametersFB.IO.DOut.T_QM2_OnTime > LTIME#30s and ParametersFB.IO.DOut.F_QM1_OnTime > LTIME#30s;
END_METHOD

METHOD ExtractFanOverride : BOOL
VAR_INPUT
	Override: BOOL;
	Speed: LREAL;
END_VAR
END_METHOD

METHOD FB_init : BOOL
VAR_INPUT
	bInitRetains : BOOL; // if TRUE, the retain variables are initialized (warm start / cold start)
	bInCopyCode : BOOL;  // if TRUE, the instance afterwards gets moved into the copy code (online change)
END_VAR
IF bInitRetains THEN
	;
END_IF
END_METHOD

METHOD Fire : BOOL
VAR_INPUT
END_VAR
Parameters.IO.DOut.F_QM2 := FALSE;
Fire := TRUE;
END_METHOD

METHOD FireAlarm : BOOL
VAR_INPUT
END_VAR
VAR_INST
END_VAR
FireAlarm := Parameters.Alarm.Active.A.FireExtract OR 
	Parameters.Alarm.Active.A.FireSupply OR
	Parameters.Alarm.Active.A.FireExtractPressure OR
	Parameters.Alarm.Active.A.FireExtractTemperature OR
	Parameters.Alarm.Active.A.FireExtractExternal;
END_METHOD

METHOD FireEnd : BOOL
VAR_INPUT
END_VAR
Parameters.IO.DOut.F_QM2 := TRUE;
END_METHOD

METHOD FireSupply : BOOL
VAR_INPUT
END_VAR
FireSupply := TRUE;
END_METHOD

METHOD FireSupplyEnd : BOOL
VAR_INPUT
END_VAR
END_METHOD

{attribute 'TcEncoding':='UTF-8'}
METHOD GetActiveStateName : string
VAR_INPUT
END_VAR
GetActiveStateName := TO_STRING(Parameters.System.Operation.State);
END_METHOD

METHOD GetCurrentExtractAirPV : LREAL
VAR_INPUT
END_VAR

IF Parameters.Regulation.ExtractAir.ControlMode =  FanControlTypes.Pressure  THEN
	GetCurrentExtractAirPV := Parameters.IO.AIn.F_BP1;
ELSE
	GetCurrentExtractAirPV := Parameters.IO.AIn.F_BF1;
END_IF
END_METHOD

METHOD GetCurrentPV : LREAL
VAR_INPUT
END_VAR
GetCurrentPV := Parameters.IO.AIn.T_BT1;
IF Parameters.Regulation.Temperature.TemperatureControlSource = TemperatureControlSources.F_BT1 THEN
	GetCurrentPV := Parameters.IO.AIn.F_BT1;
ELSIF Parameters.Regulation.Temperature.TemperatureControlSource = TemperatureControlSources.BT2 THEN
	GetCurrentPV := Parameters.IO.AIn.BT2;
END_IF
END_METHOD

METHOD GetCurrentSP : LREAL
VAR_INPUT
END_VAR
IF Parameters.Regulation.Temperature.TemperatureControlSource = TemperatureControlSources.F_BT1 THEN
	GetCurrentSP := Parameters.Regulation.Temperature.Control.SP + Parameters.Regulation.Temperature.SetPointAdjustment.Y;
ELSE
	GetCurrentSP := Parameters.Regulation.Temperature.Control.SP;
END_IF
END_METHOD

METHOD GetCurrentSupplyAirPV : LREAL
VAR_INPUT
END_VAR

IF Parameters.Regulation.SupplyAir.ControlMode =  FanControlTypes.Pressure  THEN
	GetCurrentSupplyAirPV := Parameters.IO.AIn.T_BP1;
ELSE
	GetCurrentSupplyAirPV := Parameters.IO.AIn.T_BF1;
END_IF
END_METHOD

METHOD GetFireExtractAlarms : BOOL
VAR_INPUT
END_VAR
GetFireExtractAlarms := Parameters.Alarm.Active.A.FireExtract OR
	Parameters.Alarm.Active.A.FireExtractPressure OR
	Parameters.Alarm.Active.A.FireExtractTemperature OR
	Parameters.Alarm.Active.A.FireExtractExternal;
END_METHOD

METHOD GetParameters : reference to GreenMasterBaseParameters
VAR_INPUT
END_VAR
GetParameters REF= Parameters;
END_METHOD

METHOD GetParametersFB : reference to GreenMasterBaseParametersFB
VAR_INPUT
END_VAR
GetParametersFB REF= ParametersFB;
END_METHOD

METHOD GetParametersSC : reference to SmokeControlParametersBase
VAR_INPUT
END_VAR
GetParametersSC REF= ParametersSC;
END_METHOD

METHOD GetParametersSCFB : reference to SmokeControlParametersBaseFB
VAR_INPUT
END_VAR
GetParametersSCFB REF= ParametersSCFB;
END_METHOD

METHOD GetState : SystemStates
VAR_INPUT
END_VAR
GetState := Parameters.System.Operation.State;
END_METHOD

METHOD Runnable : BOOL
VAR_INPUT
	IncludeSP: bool;
END_VAR
Runnable := ENO AND (
	NOT (Parameters.Alarm.Active.A.Freeze OR 
		Parameters.Alarm.Active.B.ExtractFan OR 
		Parameters.Alarm.Active.B.SupplyFan OR 
		Parameters.IO.AIn.F_BP1_Error OR
		Parameters.IO.AIn.T_BP1_Error)
	) AND
	(Parameters.IO.DIn.Hand OR (Parameters.IO.DIn.Auto AND (Parameters.System.Operation.TimeChannels.Q or Parameters.Regulation.NightCooling))) AND
	(ADS_Standard.Tags.Settings.RemoteStart > 0) AND
	(
		(Parameters.Regulation.ExtractAir.Control.CSP <> 0) OR
		(Parameters.Regulation.SupplyAir.Control.CSP <> 0) OR
		(NOT IncludeSP)
	);
END_METHOD

METHOD Simulate : BOOL
VAR_INPUT
	Parameters: REFERENCE TO GreenMasterBaseParameters;
	ParametersFB: REFERENCE TO GreenMasterBaseParametersFB;
END_VAR

VAR
	CurrentF_Fan: LREAL;
	CurrentT_Fan: LREAL;
END_VAR

VAR_INST
	FirstTime: BOOL;
	F_Pressure: LREAL;
	T_Pressure: LREAL;
	LastSecond: LINT;
END_VAR
IF NOT FirstTime THEN
	FirstTime := TRUE;
	Parameters.IO.DIn.Auto := TRUE;
	Parameters.IO.DIn.F_QM2_Open := TRUE;
	Parameters.IO.DIn.FireExtractAlarm := FALSE;
	Parameters.IO.DIn.FuseAlarm := FALSE;
	Parameters.IO.DIn.FireSupplyAlarm := FALSE;
	Parameters.IO.DIn.T_GQ1_Alarm := FALSE;
	Parameters.IO.DIn.F_GQ1_Alarm := FALSE;
	Parameters.IO.AIn.BT1 := 10;
	Parameters.IO.AIn.BT2 := 20;
	Parameters.IO.AIn.F_BF1 := 0;
	Parameters.IO.AIn.F_BP1 := 0;
	Parameters.IO.AIn.F_BP2 := 0;
	Parameters.IO.AIn.F_BP3 := 0;
	Parameters.IO.AIn.F_BT1 := 20;
	Parameters.IO.AIn.F_BT2 := 20;
	Parameters.IO.AIn.H_BT1 := 20;
	Parameters.IO.AIn.T_BF1 := 0;
	Parameters.IO.AIn.T_BP1 := 0;
	Parameters.IO.AIn.T_BP2 := 0;
	Parameters.IO.AIn.T_BT1 := 18;
	Parameters.IO.AIn.T_BT2 := 10;
	Parameters.IO.AIn.T_BT3 := 20;
END_IF
IF Globals.SecondsCounter <> LastSecond THEN	
	CurrentT_Fan := Parameters.IO.AOut.T_GQ1;
	CurrentF_Fan := Parameters.IO.AOut.F_GQ1;
	(*
	IF Main.ParallelUnits.EN THEN
		CurrentT_Fan := LIMIT(0, CurrentT_Fan + Main.ParallelUnits.RemoteStatusData.RemoteStatus.SupplyFanSpeed, 2); 
		CurrentF_Fan := LIMIT(0, CurrentF_Fan + Main.ParallelUnits.RemoteStatusData.RemoteStatus.ExtractFanSpeed, 2); 
	END_IF
	*)
	Parameters.IO.DIn.H_GP1_Running := Parameters.IO.DOut.H_GP1;
	T_Pressure := ((1 + CurrentT_Fan) * (1 + CurrentT_Fan) - 1) * 150 - 1;
	Parameters.IO.AIn.T_BP1 := T_Pressure;
	F_Pressure := ((1 + CurrentF_Fan) * (1 + CurrentF_Fan) - 1) * 150 - 1;
	Parameters.IO.AIn.F_BP1 := F_Pressure;
	Parameters.IO.DIn.F_QM2_Closed := ParametersFB.IO.DOut.F_QM2_OnTime < LTIME#5S; 
	Parameters.IO.DIn.F_QM2_Open := ParametersFB.IO.DOut.F_QM2_OnTime > LTIME#30S; 
	LastSecond := Globals.SecondsCounter;
END_IF
END_METHOD

METHOD StateTime : LTIME
VAR_INPUT
END_VAR
StateTime := LTIME() - StateStartTime;
END_METHOD

METHOD SupplyFanOverride : BOOL
VAR_INPUT
	Override: BOOL;
	Speed: LREAL;
END_VAR
END_METHOD

METHOD SystemStateST : BOOL
VAR_IN_OUT
	Parameters: GreenMasterBaseParameters;
END_VAR
VAR_INPUT
END_VAR
VAR_INST
	SystemStateSTInitDone: BOOL;
	CurrentStateTime: LTIME;
END_VAR
VAR_INST
	State: REFERENCE TO SystemStates;
	NextState: SystemStates;	
END_VAR
VAR
	LogStr: string;
END_VAR
State REF= Parameters.System.Operation.State;
IF NOT SystemStateSTInitDone THEN
	SystemStateStarted();
	State := SystemStates.Idle;	
	SystemStateSTInitDone := TRUE;
END_IF

IF NextState <> State THEN
	LogStr := 'Entering state ';
	LogStr := Concat(LogStr, TO_STRING(NextState));
	Main.EventLog.LogEvent(Message := LogStr, Kind := EventTypes.Information);
	SystemStateStarted();
	// Entry state logic
	CASE NextState OF

		SystemStates.Start:
			;
			
		SystemStates.Idle:
			SystemStateVentilation := FALSE;
			Parameters.IO.DOut.F_QM1 := FALSE;
			Parameters.IO.DOut.T_QM2 := FALSE;
			Parameters.IO.AOut.F_QN1 := 0;
			Parameters.IO.AOut.F_GQ1 := 0;
			Parameters.IO.AOut.T_GQ1 := 0;
			Parameters.IO.DOut.T_QM1_1 := FALSE;
			Parameters.IO.DOut.T_QM1_2 := FALSE;
			Parameters.IO.DOut.T_QM1_3 := FALSE;
			Parameters.IO.DOut.T_QM1_4 := FALSE;
			Parameters.IO.DOut.T_QM1_5 := FALSE;
			Parameters.IO.DOut.T_QM1_6 := FALSE;
			Parameters.IO.AOut.F_GQ1 := 0;
			Parameters.IO.AOut.T_GQ1 := 0;
			ExtractFanOverride(FALSE, 0);
			SupplyFanOverride(FALSE, 0);
			
		SystemStates.OpenDampers:
			Parameters.IO.AOut.F_QN1 := 0;
			SystemStateVentilation := TRUE;

		SystemStates.StartupHeatRecovery:
			;
		SystemStates.Run:
			;

		SystemStates.FireHandling:
			SystemStateVentilation := FALSE;

		SystemStates.FireExhaust:
			Parameters.IO.AOut.F_QN1 := 0;
			Parameters.IO.DOut.F_QM1 := FALSE;
			Parameters.IO.DOut.F_QM2 := NOT Parameters.Regulation.ExtractAir.FireExhaust.EN;
			Parameters.IO.DOut.T_QM2 := Parameters.Regulation.SupplyAir.FireSupply.EN;
			Parameters.IO.DOut.T_QM1_1 := Parameters.Regulation.SupplyAir.FireSupply.EN;
			Parameters.IO.DOut.T_QM1_2 := Parameters.Regulation.SupplyAir.FireSupply.EN;
			Parameters.IO.DOut.T_QM1_3 := Parameters.Regulation.SupplyAir.FireSupply.EN;
			Parameters.IO.DOut.T_QM1_4 := Parameters.Regulation.SupplyAir.FireSupply.EN;
			Parameters.IO.DOut.T_QM1_5 := Parameters.Regulation.SupplyAir.FireSupply.EN;
			Parameters.IO.DOut.T_QM1_6 := Parameters.Regulation.SupplyAir.FireSupply.EN;
			Fire();
				
		SystemStates.FireSupply:
			FireSupply();	
			Parameters.IO.AOut.F_QN1 := 0;
			Parameters.IO.DOut.F_QM1 := FALSE;
			Parameters.IO.DOut.F_QM2 := NOT Parameters.Regulation.ExtractAir.FireExhaust.EN;
			Parameters.IO.DOut.T_QM2 := Parameters.Regulation.SupplyAir.FireSupply.EN;
			Parameters.IO.DOut.T_QM1_1 := Parameters.Regulation.SupplyAir.FireSupply.EN;
			Parameters.IO.DOut.T_QM1_2 := Parameters.Regulation.SupplyAir.FireSupply.EN;
			Parameters.IO.DOut.T_QM1_3 := Parameters.Regulation.SupplyAir.FireSupply.EN;
			Parameters.IO.DOut.T_QM1_4 := Parameters.Regulation.SupplyAir.FireSupply.EN;
			Parameters.IO.DOut.T_QM1_5 := Parameters.Regulation.SupplyAir.FireSupply.EN;
			Parameters.IO.DOut.T_QM1_6 := Parameters.Regulation.SupplyAir.FireSupply.EN;

		SystemStates.Ventilate:
			;

		SystemStates.Exercise:
			SystemStateVentilation := FALSE;
	END_CASE;
end_if;

State := NextState;
CurrentStateTime := StateTime();

// Do while in state logic
CASE State OF

	SystemStates.Start:
		;
		
	SystemStates.Idle:
		Parameters.System.Operation.Mode := SystemStatesRunMode.Off;
		Parameters.IO.AOut.F_QN1 := 0;
		IF StateTime() > LTIME#30S THEN
			CloseDampers();
		END_IF
		
	SystemStates.OpenDampers:
		Parameters.IO.DOut.F_QM1 := TRUE;		
		Parameters.IO.DOut.F_QM2 := TRUE;
		Parameters.IO.DOut.R_QM1 := FALSE;
		ExtractFanOverride(TRUE, 0);
		SupplyFanOverride(TRUE, 0);

	SystemStates.StartupHeatRecovery:
		IF StateTime() > TO_LTIME(Parameters.System.Operation.ExhaustFanStartupDelay) THEN
			ExtractFanOverride(TRUE, Parameters.Regulation.ExtractAir.StartupFanSpeed);
			//Parameters.IO.AOut.F_GQ1 := Parameters.Regulation.ExtractAir.StartupFanSpeed;			
			Parameters.IO.DOut.T_QM2 := TRUE;
			Parameters.IO.DOut.T_QM1_1 := TRUE;
			Parameters.IO.DOut.T_QM1_2 := TRUE;
			Parameters.IO.DOut.T_QM1_3 := TRUE;
			Parameters.IO.DOut.T_QM1_4 := TRUE;
			Parameters.IO.DOut.T_QM1_5 := TRUE;
			Parameters.IO.DOut.T_QM1_6 := TRUE;
		END_IF
		IF StateTime() > TO_LTIME(Parameters.System.Operation.SupplyFanStartupDelay) THEN
			SupplyFanOverride(TRUE, Parameters.Regulation.SupplyAir.StartupFanSpeed);
		END_IF
		
	SystemStates.Run:
		
		ExtractFanOverride(FALSE, 0);
		SupplyFanOverride(FALSE, 0);
		Parameters.System.Operation.Mode := SystemStatesRunMode.LowSpeed;
		ColdRecyclingHysteresis(	EN := Parameters.Regulation.Temperature.ColdRecycling.EN, 
									Value := Parameters.IO.AIn.F_BT1, 
									LimitValue := Parameters.Regulation.CompensationTemperature + Parameters.Regulation.Temperature.ColdRecycling.Offset, 
									Offset := Parameters.Regulation.Temperature.ColdRecycling.Hysteresis);

	SystemStates.FireHandling:
		;

	SystemStates.FireExhaust:
		Fire();
		Parameters.IO.DOut.F_QM2 := NOT Parameters.Regulation.ExtractAir.FireExhaust.EN;
		Parameters.IO.DOut.T_QM2 := Parameters.Regulation.SupplyAir.FireSupply.EN;
		Parameters.IO.DOut.T_QM1_1 := Parameters.Regulation.SupplyAir.FireSupply.EN;
		Parameters.IO.DOut.T_QM1_2 := Parameters.Regulation.SupplyAir.FireSupply.EN;
		Parameters.IO.DOut.T_QM1_3 := Parameters.Regulation.SupplyAir.FireSupply.EN;
		Parameters.IO.DOut.T_QM1_4 := Parameters.Regulation.SupplyAir.FireSupply.EN;
		Parameters.IO.DOut.T_QM1_5 := Parameters.Regulation.SupplyAir.FireSupply.EN;
		Parameters.IO.DOut.T_QM1_6 := Parameters.Regulation.SupplyAir.FireSupply.EN;
			
	SystemStates.FireSupply:
		FireSupply();
		Parameters.IO.DOut.F_QM2 := NOT Parameters.Regulation.ExtractAir.FireExhaust.EN;
		Parameters.IO.DOut.T_QM2 := Parameters.Regulation.SupplyAir.FireSupply.EN;
		Parameters.IO.DOut.T_QM1_1 := Parameters.Regulation.SupplyAir.FireSupply.EN;
		Parameters.IO.DOut.T_QM1_2 := Parameters.Regulation.SupplyAir.FireSupply.EN;
		Parameters.IO.DOut.T_QM1_3 := Parameters.Regulation.SupplyAir.FireSupply.EN;
		Parameters.IO.DOut.T_QM1_4 := Parameters.Regulation.SupplyAir.FireSupply.EN;
		Parameters.IO.DOut.T_QM1_5 := Parameters.Regulation.SupplyAir.FireSupply.EN;
		Parameters.IO.DOut.T_QM1_6 := Parameters.Regulation.SupplyAir.FireSupply.EN;

	SystemStates.Ventilate:
		;

	SystemStates.Exercise:
		;
end_case;

// Transitions

CASE State OF

	SystemStates.None:
		NextState := SystemStates.Start;
 
	SystemStates.Start:
		NextState := SystemStates.Idle;
		
	SystemStates.Idle:
		if FireAlarm() then
			NextState := SystemStates.FireHandling;
		end_if;
		IF Runnable(IncludeSP := TRUE) THEN
			NextState := SystemStates.OpenDampers;
		end_if;
		
	SystemStates.OpenDampers:
		if FireAlarm() then
			NextState := SystemStates.FireHandling;
		end_if;
		IF StateTime() > TO_LTIME(Parameters.System.Operation.StartupDamperWaitTime) THEN
			NextState := SystemStates.StartupHeatRecovery;
		end_if;
		IF NOT Runnable(IncludeSP := TRUE) THEN
			NextState := SystemStates.Idle;
		end_if;
		IF SmokeControl.Exercising OR Main.GreenMaster.ExerciseF_QM2.Exercising THEN
			NextState := SystemStates.Exercise;
		end_if;

	SystemStates.StartupHeatRecovery:
		if FireAlarm() then
			NextState := SystemStates.FireHandling;
		end_if;
		IF NOT Runnable(IncludeSP := TRUE) THEN
			NextState := SystemStates.Idle;
		END_IF;
		IF StateTime() > TO_LTIME(Parameters.System.Operation.StartupHeatRecoveryTime) THEN
			NextState := SystemStates.Run;
		END_IF;
		IF SmokeControl.Exercising OR Main.GreenMaster.ExerciseF_QM2.Exercising THEN
			NextState := SystemStates.Exercise;
		end_if;
		
	SystemStates.Run:
		if FireAlarm() then
			NextState := SystemStates.FireHandling;
		end_if;
			
		IF NOT Runnable(IncludeSP := TRUE) THEN
			NextState := SystemStates.PostRun;
		end_if;
		IF SmokeControl.Exercising OR Main.GreenMaster.ExerciseF_QM2.Exercising THEN
			NextState := SystemStates.Exercise;
		end_if;

	SystemStates.PostRun:
		if FireAlarm() then
			NextState := SystemStates.FireHandling;
		end_if;
		IF NOT Runnable(IncludeSP := TRUE) THEN
			NextState := SystemStates.Idle;
		end_if;
		IF StateTime() > TO_LTIME(Parameters.System.Operation.PostVentilationTime) THEN
			NextState := SystemStates.Idle;
		end_if;
		
	SystemStates.FireHandling:
		FireAlarm();
		IF Parameters.Alarm.Active.A.FireSupply AND NOT GetFireExtractAlarms() THEN
			NextState := SystemStates.FireSupply;
		ELSIF GetFireExtractAlarms() THEN
			NextState := SystemStates.FireExhaust;
		ELSE
			NextState := SystemStates.FireHandlingExit;			
		END_IF;
		
	SystemStates.FireHandlingExit:
		FireAlarm();
		NextState := SystemStates.Idle;

	SystemStates.FireExhaust:
		FireAlarm();
		IF NOT Parameters.Alarm.Active.A.FireSupply AND NOT GetFireExtractAlarms() THEN
			NextState := SystemStates.Ventilate;
		end_if;
		IF Parameters.Alarm.Active.A.FireSupply AND NOT GetFireExtractAlarms() THEN
			NextState := SystemStates.FireSupply;
		end_if;
			
	SystemStates.FireSupply:
		FireAlarm();
		IF GetFireExtractAlarms() THEN
			NextState := SystemStates.FireExhaust;
		end_if;
		IF NOT Parameters.Alarm.Active.A.FireSupply THEN
			NextState := SystemStates.FireHandlingExit;
		end_if;

	SystemStates.Ventilate:
		FireAlarm();
		IF NOT Parameters.Alarm.Active.A.FireSupply AND GetFireExtractAlarms() THEN
			NextState := SystemStates.FireExhaust;
		END_IF;
		IF Parameters.Alarm.Active.A.FireSupply THEN
			NextState := SystemStates.FireSupply;
		END_IF
		IF TRUE (* StateTime() > Parameters.System.Operation.PostFireVentilationTime *) THEN
			NextState := SystemStates.FireHandlingExit;
		END_IF;
		
	SystemStates.Exercise:
		FireAlarm();
		IF NOT (SmokeControl.Exercising OR Main.GreenMaster.ExerciseF_QM2.Exercising)  THEN
			NextState := SystemStates.Idle;		
		END_IF;
END_CASE;

IF NextState <> State THEN

	// Exit state logic
	CASE State OF

		SystemStates.Start:
			;
			
		SystemStates.Idle:
			;
			
		SystemStates.OpenDampers:
			;

		SystemStates.StartupHeatRecovery:
			//OvrTemperatureControl := TRUE;	
			
		SystemStates.Run:
			;

		SystemStates.FireHandling:
			;

		SystemStates.FireExhaust:
			FireEnd();
				
		SystemStates.FireSupply:
			FireSupplyEnd();

		SystemStates.Ventilate:
			;

	end_case;
end_if;
END_METHOD

METHOD SystemStateStarted : BOOL
VAR_INPUT
END_VAR
StateStartTime := LTIME();
END_METHOD

METHOD Update : BOOL
VAR_INPUT
	DO_: REFERENCE TO GreenMasterDO_Base;
	AO: REFERENCE TO GreenMasterAO_Base;
END_VAR

VAR_INST
	FirstTime: BOOL;
END_VAR
IF NOT FirstTime THEN
	FirstTime := TRUE;
END_IF

FireAlarmExtractAirTemperatureHysteresis(Value := Parameters.IO.AIn.F_BT1,
	LimitValue := Parameters.Alarm.Limits.A.FireExtractTemperature,
	Offset := 1);
	
FireAlarmExtractAirPressureTemperatureHysteresis(Value := Parameters.IO.AIn.F_BT1,
	LimitValue := Parameters.Alarm.Limits.A.FireExtractPressureTemperature,
	Offset := 1);
	
FireAlarmExtractAirPressureHysteresis(Value := Parameters.IO.AIn.F_BP2,
	LimitValue := Parameters.Alarm.Limits.A.FireExtractPressure,
	Offset := 10);
	
Parameters.Alarm.Status.A.FireExtractTemperature := FireAlarmExtractAirTemperatureHysteresis.Above;
Parameters.Alarm.Status.A.FireExtractPressure := FireAlarmExtractAirPressureTemperatureHysteresis.Above AND
	FireAlarmExtractAirPressureHysteresis.Above;

IF Reverse_C_QN1 THEN
	C_QN1_Low := 1;
	C_QN1_High := 0;
ELSE
	C_QN1_Low := 0;
	C_QN1_High := 1;
END_IF

UpdateIO(DO_ := DO_, AO := AO);

SystemStateST(Parameters := Parameters);

ParametersFB(GreenMaster := THIS^);
END_METHOD

METHOD UpdateIO : BOOL
VAR_INPUT
	DO_: REFERENCE TO GreenMasterDO_Base;
	AO: REFERENCE TO GreenMasterAO_Base;
END_VAR
ParametersFB.IO.AIn();
ParametersFB.IO.AOut();
ParametersFB.IO.DIn();
ParametersFB.IO.DOut(DOut := Parameters.IO.DOut);

ParametersFB.IO.AIn.Update(AI := AI, AI2 := AI2, Parameters := Parameters);
ParametersFB.IO.AOut.Update(AO := AO, Parameters  := Parameters, AOut := Parameters.IO.AOut);
ParametersFB.IO.DIn.Update(DI := DI, Parameters := Parameters, DIn := Parameters.IO.DIn);
ParametersFB.IO.DOut.Update(DO_ := DO_, Parameters := Parameters, EnableWriteDampers := EnableFansAndDampers);
END_METHOD

END_FUNCTION_BLOCK

// ---- DUTs/Parameters/GreenMasterBaseParametersFB.TcPOU
FUNCTION_BLOCK GreenMasterBaseParametersFB
VAR_IN_OUT
	GreenMaster: GreenMasterBase;
END_VAR
VAR_INPUT
END_VAR
VAR_OUTPUT
	System: SystemParametersFB;
	Regulation: RegulationParametersFB;
	//Alarm: AlarmParametersFB;
	IO: IoParametersFB;
	Simulation: SimulationFB;
END_VAR
VAR
END_VAR

System(ParametersFB := THIS^, Parameters := GreenMaster.GetParameters(), System := GreenMaster.GetParameters().System);
Regulation(ParametersFB := THIS^, Parameters := GreenMaster.GetParameters(), Regulation := GreenMaster.GetParameters().Regulation);
IO(GreenMaster := GreenMaster, ParametersFB := THIS^, Parameters := GreenMaster.GetParameters());

METHOD GetGreenMaster : REFERENCE TO GreenMasterBase
VAR_INPUT
END_VAR
GetGreenMaster REF= GreenMaster;
END_METHOD

END_FUNCTION_BLOCK

// ---- DUTs/Parameters/System/SystemParametersFB.TcPOU
(* This is a comment 1
	with multiple lines
*)
FUNCTION_BLOCK SystemParametersFB
VAR_IN_OUT
	Parameters: GreenMasterBaseParameters;
	ParametersFB: GreenMasterBaseParametersFB;
	System: SystemParameters;
END_VAR
VAR_INPUT
END_VAR
VAR_OUTPUT
	Exercise: ExerciseParametersFB;
	Operation: OperationParametersFB;
END_VAR
VAR
	LastSecondsCounter: lint;
END_VAR

Exercise(Parameters := Parameters, ParametersFB := ParametersFB);
System.Operation.ENO := System.Operation.State > SystemStates.Idle;
Operation(Parameters := Parameters, ParametersFB := ParametersFB);
IF (Globals.SecondsCounter - LastSecondsCounter) > 10 THEN
	LastSecondsCounter := Globals.SecondsCounter;
	
	System.Operation.TimeChannels.Q :=
		System.Operation.TimeChannels.TC01.Q OR
		System.Operation.TimeChannels.TC02.Q OR
		System.Operation.TimeChannels.TC03.Q OR
		System.Operation.TimeChannels.TC04.Q OR
		System.Operation.TimeChannels.TC05.Q OR
		System.Operation.TimeChannels.TC06.Q OR
		System.Operation.TimeChannels.TC07.Q OR
		System.Operation.TimeChannels.TC11.Q OR
		System.Operation.TimeChannels.TC12.Q OR
		System.Operation.TimeChannels.TC13.Q OR
		System.Operation.TimeChannels.TC14.Q OR
		System.Operation.TimeChannels.TC15.Q OR
		System.Operation.TimeChannels.TC16.Q OR
		System.Operation.TimeChannels.TC17.Q OR
		System.Operation.TimeChannels.TC21.Q OR
		System.Operation.TimeChannels.TC22.Q OR
		System.Operation.TimeChannels.TC23.Q OR
		System.Operation.TimeChannels.TC24.Q OR
		System.Operation.TimeChannels.TC25.Q OR
		System.Operation.TimeChannels.TC26.Q OR
		System.Operation.TimeChannels.TC27.Q;
	System.Operation.TimeChannels.HighSpeed := 
		(System.Operation.TimeChannels.TC01.Q AND (System.Operation.TimeChannels.TC01.Speed = 2)) OR
		(System.Operation.TimeChannels.TC02.Q AND (System.Operation.TimeChannels.TC02.Speed = 2)) OR
		(System.Operation.TimeChannels.TC03.Q AND (System.Operation.TimeChannels.TC03.Speed = 2)) OR
		(System.Operation.TimeChannels.TC04.Q AND (System.Operation.TimeChannels.TC04.Speed = 2)) OR
		(System.Operation.TimeChannels.TC05.Q AND (System.Operation.TimeChannels.TC05.Speed = 2)) OR
		(System.Operation.TimeChannels.TC06.Q AND (System.Operation.TimeChannels.TC06.Speed = 2)) OR
		(System.Operation.TimeChannels.TC07.Q AND (System.Operation.TimeChannels.TC07.Speed = 2)) OR
		(System.Operation.TimeChannels.TC11.Q AND (System.Operation.TimeChannels.TC11.Speed = 2)) OR
		(System.Operation.TimeChannels.TC12.Q AND (System.Operation.TimeChannels.TC12.Speed = 2)) OR
		(System.Operation.TimeChannels.TC13.Q AND (System.Operation.TimeChannels.TC13.Speed = 2)) OR
		(System.Operation.TimeChannels.TC14.Q AND (System.Operation.TimeChannels.TC14.Speed = 2)) OR
		(System.Operation.TimeChannels.TC15.Q AND (System.Operation.TimeChannels.TC15.Speed = 2)) OR
		(System.Operation.TimeChannels.TC16.Q AND (System.Operation.TimeChannels.TC16.Speed = 2)) OR
		(System.Operation.TimeChannels.TC17.Q AND (System.Operation.TimeChannels.TC17.Speed = 2)) OR
		(System.Operation.TimeChannels.TC21.Q AND (System.Operation.TimeChannels.TC21.Speed = 2)) OR
		(System.Operation.TimeChannels.TC22.Q AND (System.Operation.TimeChannels.TC22.Speed = 2)) OR
		(System.Operation.TimeChannels.TC23.Q AND (System.Operation.TimeChannels.TC23.Speed = 2)) OR
		(System.Operation.TimeChannels.TC24.Q AND (System.Operation.TimeChannels.TC24.Speed = 2)) OR
		(System.Operation.TimeChannels.TC25.Q AND (System.Operation.TimeChannels.TC25.Speed = 2)) OR
		(System.Operation.TimeChannels.TC26.Q AND (System.Operation.TimeChannels.TC26.Speed = 2)) OR
		(System.Operation.TimeChannels.TC27.Q AND (System.Operation.TimeChannels.TC27.Speed = 2));
END_IF

END_FUNCTION_BLOCK

// ---- DUTs/Parameters/System/Exercise/ExerciseParametersFB.TcPOU
FUNCTION_BLOCK ExerciseParametersFB
VAR_IN_OUT
	Parameters: GreenMasterBaseParameters;
	ParametersFB: GreenMasterBaseParametersFB;
END_VAR
VAR_INPUT
END_VAR
VAR_OUTPUT
	CirculationPumps: ExerciseCirculationPumpsParametersFB;
	FireBypassDamper: ExerciseFireBypassDamperParametersFB;
END_VAR
VAR
	LA02_P1_EXTC: TimeChannel1CH;
	LA02_P2_EXTC: TimeChannel1CH;
	LA02_SV_ST_EXTC: TimeChannel1CH;
	ExerciseState: INT;	
END_VAR

ParametersFB.System.Exercise.CirculationPumps();
ParametersFB.System.Exercise.FireBypassDamper();
//Parameters.System.Exercise.ExternalFireControl();

(*
LA02_P1_EXTC(Settings := ADS_CTH.Tags.Settings.LA02_P1X_TC);
LA02_P2_EXTC(Settings := ADS_CTH.Tags.Settings.LA02_P2X_TC);
Globals.IO.DOut.DO01 := LA02_P1_EXTC.Q;
Globals.IO.DOut.DO16 := LA02_P2_EXTC.Q;
LA02_SV_ST_EXTC(Settings := ADS_CTH.Tags.Settings.LA02_SX_TC);
IF LA02_SV_ST_EXTC.Q THEN
	CASE ExerciseState OF
		1:
			Globals.IO.AOut.AO01 := 0;
			Globals.IO.AOut.AO05 := 0;
			Globals.IO.DOut.DO04 := FALSE;
			Globals.IO.DOut.DO05 := FALSE;
		2:
			Globals.IO.AOut.AO01 := 32767;
			Globals.IO.AOut.AO05 := 32767;
			Globals.IO.DOut.DO04 := TRUE;
			Globals.IO.DOut.DO05 := TRUE;
		3:
			ExerciseState := 0;
	END_CASE
END_IF
*)

END_FUNCTION_BLOCK

// ---- DUTs/Parameters/System/Exercise/ExerciseCirculationPumpsParametersFB.TcPOU
FUNCTION_BLOCK ExerciseCirculationPumpsParametersFB
VAR_INPUT
END_VAR
VAR_OUTPUT
END_VAR
VAR
END_VAR

END_FUNCTION_BLOCK

// ---- DUTs/Parameters/System/Exercise/ExerciseFireBypassDamperParametersFB.TcPOU
FUNCTION_BLOCK ExerciseFireBypassDamperParametersFB
VAR_INPUT
END_VAR
VAR_OUTPUT
END_VAR
VAR
END_VAR

END_FUNCTION_BLOCK

// ---- DUTs/Utilities/TimeChannel1CH.TcPOU
FUNCTION_BLOCK TimeChannel1CH
VAR_INPUT
	Data: REFERENCE TO TimeChannel1CH_Data;
END_VAR
VAR_OUTPUT
END_VAR
VAR
	CurrentDay: WORD; // $(skip)
	DayMatch: BOOL; // $(skip)
	LocalSystemTime: FB_LocalSystemTime; // $(skip)
	IsOnTime: BOOL; // $(skip)
	MinuteOfDay: WORD; // $(skip)
	StartMinuteOfDay: WORD; // $(skip)
	EndMinuteOfDay: WORD; // $(skip)
	OnHour           : UINT;	(* Hour value of the switch-on time on the day $(skip) *)
	OnMinute         : UINT;	(* Minute value of the switch-on time on the day $(skip) *)
	OffHour          : UINT;	(* Hour value of the switch-off time on the day $(skip) *)
	OffMinute        : UINT;	(* Minute value of the switch-off time on the day $(skip) *)
END_VAR

Data.Error := FALSE;
OnHour := Data.OnTime / 100;
OnMinute := Data.OnTime MOD 100;
OffHour := Data.OffTime / 100;
OffMinute := Data.OffTime MOD 100;
LocalSystemTime(bEnable := TRUE);
IF Data.EN AND (NOT Data.Error) THEN
	IF LocalSystemTime.bValid THEN	
		CurrentDay := F_GetDayOfWeek(in := NowDT()); 
		DayMatch := Data.Day = TimerDays.AllDays OR (TO_WORD(Data.Day) = CurrentDay - 1);
		IF OnHour = OffHour AND OnMinute = OffMinute THEN
			Data.Q := FALSE;
		ELSE
			MinuteOfDay := LocalSystemTime.systemTime.wHour * 60 + LocalSystemTime.systemTime.wMinute;
			StartMinuteOfDay := OnHour * 60 + OnMinute;
			EndMinuteOfDay := OffHour * 60 + OffMinute;
			IsOnTime := MinuteOfDay >= StartMinuteOfDay AND MinuteOfDay < EndMinuteOfDay;
			Data.Q := DayMatch AND IsOnTime;				
			IF Data.Q AND Data.SingleShot THEN
				Data.EN := FALSE;
			END_IF
		END_IF
		Data.ENO := TRUE;
	ELSE
		Data.Q := FALSE;
		Data.ENO := FALSE;
	END_IF
ELSE
	Data.Q := FALSE;
	Data.ENO := FALSE;
END_IF

END_FUNCTION_BLOCK

// ---- DUTs/Utilities/NowDT.TcPOU
FUNCTION NowDT : DT
VAR_INPUT
END_VAR
VAR
	timeAsFileTime: T_FILETIME;
END_VAR
VAR_STAT
	fbSystemTime: GETSYSTEMTIME;
END_VAR

fbSystemTime(
	timeLoDW =>timeAsFileTime.dwLowDateTime,
	timeHiDW =>timeAsFileTime.dwHighDateTime 
);
NowDT := FILETIME_TO_DT( timeAsFileTime );

END_FUNCTION

// ---- DUTs/Parameters/System/Operation/OperationParametersFB.TcPOU
FUNCTION_BLOCK OperationParametersFB
VAR_INPUT
	Parameters: REFERENCE TO GreenMasterBaseParameters;
	ParametersFB: REFERENCE TO GreenMasterBaseParametersFB;
END_VAR
VAR_OUTPUT
	TimeChannelsParametersFB: TimeChannelParametersFB;
END_VAR
VAR
END_VAR

TimeChannelsParametersFB(Parameters := Parameters, ParametersFB := ParametersFB);

END_FUNCTION_BLOCK

// ---- DUTs/Parameters/System/Operation/TimeChannelParametersFB.TcPOU
FUNCTION_BLOCK TimeChannelParametersFB
VAR_INPUT
	Parameters: REFERENCE TO GreenMasterBaseParameters;
	ParametersFB: REFERENCE TO GreenMasterBaseParametersFB;
END_VAR
VAR_OUTPUT
END_VAR
VAR
	TC01: TimeChannel1CH;
	TC02: TimeChannel1CH;
	TC03: TimeChannel1CH;
	TC04: TimeChannel1CH;
	TC05: TimeChannel1CH;
	TC06: TimeChannel1CH;
	TC07: TimeChannel1CH;
	TC11: TimeChannel1CH;
	TC12: TimeChannel1CH;
	TC13: TimeChannel1CH;
	TC14: TimeChannel1CH;
	TC15: TimeChannel1CH;
	TC16: TimeChannel1CH;
	TC17: TimeChannel1CH;
	TC21: TimeChannel1CH;
	TC22: TimeChannel1CH;
	TC23: TimeChannel1CH;
	TC24: TimeChannel1CH;
	TC25: TimeChannel1CH;
	TC26: TimeChannel1CH;
	TC27: TimeChannel1CH;
END_VAR

TC01(Data := Parameters.System.Operation.TimeChannels.TC01);
TC02(Data := Parameters.System.Operation.TimeChannels.TC02);
TC03(Data := Parameters.System.Operation.TimeChannels.TC03);
TC04(Data := Parameters.System.Operation.TimeChannels.TC04);
TC05(Data := Parameters.System.Operation.TimeChannels.TC05);
TC06(Data := Parameters.System.Operation.TimeChannels.TC06);
TC07(Data := Parameters.System.Operation.TimeChannels.TC07);

TC11(Data := Parameters.System.Operation.TimeChannels.TC11);
TC12(Data := Parameters.System.Operation.TimeChannels.TC12);
TC13(Data := Parameters.System.Operation.TimeChannels.TC13);
TC14(Data := Parameters.System.Operation.TimeChannels.TC14);
TC15(Data := Parameters.System.Operation.TimeChannels.TC15);
TC16(Data := Parameters.System.Operation.TimeChannels.TC16);
TC17(Data := Parameters.System.Operation.TimeChannels.TC17);

TC21(Data := Parameters.System.Operation.TimeChannels.TC21);
TC22(Data := Parameters.System.Operation.TimeChannels.TC22);
TC23(Data := Parameters.System.Operation.TimeChannels.TC23);
TC24(Data := Parameters.System.Operation.TimeChannels.TC24);
TC25(Data := Parameters.System.Operation.TimeChannels.TC25);
TC26(Data := Parameters.System.Operation.TimeChannels.TC26);
TC27(Data := Parameters.System.Operation.TimeChannels.TC27);

END_FUNCTION_BLOCK

// ---- DUTs/Parameters/Regulation/RegulationParametersFB.TcPOU
FUNCTION_BLOCK RegulationParametersFB
VAR_IN_OUT
	Parameters: GreenMasterBaseParameters;
	ParametersFB: GreenMasterBaseParametersFB;
	Regulation: RegulationParameters;
END_VAR
VAR_INPUT
END_VAR
VAR_OUTPUT
	SupplyAir: AirParametersFB;
	ExtractAir: AirParametersFB;
	Temperature: TemperatureControlParametersFB;
END_VAR
VAR
	CurrentMaxFlow: LREAL;
	NightCoolingHysteresis: Hysteresis;
END_VAR

SupplyAir(Parameters := Parameters, ParametersFB := ParametersFB, AirParameters := Regulation.SupplyAir);
ExtractAir(Parameters := Parameters, ParametersFB := ParametersFB, AirParameters := Regulation.ExtractAir);
Temperature(Parameters := Parameters, ParametersFB := ParametersFB, Temperature := Parameters.Regulation.Temperature);

IF __ISVALIDREF(ParametersFB.GetGreenMaster()) THEN
	Regulation.Temperature.Control.PV := ParametersFB.GetGreenMaster().GetCurrentPV();
	Regulation.SupplyAir.Control.PV := ParametersFB.GetGreenMaster().GetCurrentSupplyAirPV();
	Regulation.ExtractAir.Control.PV := ParametersFB.GetGreenMaster().GetCurrentExtractAirPV();
END_IF

CASE Regulation.TemperatureCompensationSource OF
	TemperatureCompensationSources.Auto:
		Regulation.CompensationTemperature := Parameters.IO.AIn.BT1;
		IF (NOT Parameters.IO.AIn.BT1_EN) OR Parameters.IO.AIn.BT1_Error THEN
			Regulation.CompensationTemperature := Parameters.IO.AIn.T_BT2;
			Regulation.CurrentTemperatureCompensationSource := TemperatureCompensationSources.T_BT2;
		ELSE
			Regulation.CurrentTemperatureCompensationSource := TemperatureCompensationSources.BT1;			
		END_IF;
	TemperatureCompensationSources.BT1:
		Regulation.CurrentTemperatureCompensationSource := TemperatureCompensationSources.BT1;
		Regulation.CompensationTemperature := Parameters.IO.AIn.BT1;
	TemperatureCompensationSources.T_BT2:
		Regulation.CurrentTemperatureCompensationSource := TemperatureCompensationSources.T_BT2;
		Regulation.CompensationTemperature := Parameters.IO.AIn.T_BT2;
END_CASE
Regulation.SupplyAir.Flow := Parameters.IO.AIn.T_BF1;
Regulation.ExtractAir.Flow := Parameters.IO.AIn.F_BF1;
Regulation.SupplyAir.Power := Main.GreenMaster.AI2.T_CurrentPower;
Regulation.ExtractAir.Power := Main.GreenMaster.AI2.F_CurrentPower;
Regulation.SupplyAir.Speed := Main.GreenMaster.AI2.T_CurrentSpeed;
Regulation.ExtractAir.Speed := Main.GreenMaster.AI2.F_CurrentSpeed;
Regulation.SupplyAir.PressureRise := Parameters.IO.AIn.T_BF1;
Regulation.ExtractAir.PressureRise := Parameters.IO.AIn.F_BF1;
CurrentMaxFlow := MAX(Regulation.ExtractAir.Flow, Regulation.SupplyAir.Flow);
IF CurrentMaxFlow <> 0 THEN
	Regulation.SystemSpecificFanPower := (Regulation.ExtractAir.Power + Regulation.SupplyAir.Power) / CurrentMaxFlow;	
ELSE
	Regulation.SystemSpecificFanPower := 0;
END_IF
IF (Regulation.SupplyAir.PressureRise + Regulation.ExtractAir.PressureRise) <> 0 THEN
	Regulation.SystemEfficiency := (Regulation.SupplyAir.SpecificFanPower + Regulation.ExtractAir.SpecificFanPower) / ((Regulation.SupplyAir.PressureRise + Regulation.ExtractAir.PressureRise) / 1000);
ELSE
	Regulation.SystemEfficiency := 0;	
END_IF

IF Regulation.ApplyAbsoluteSetPointCurves <> Regulation.LastApplyAbsoluteSetPointCurves THEN
	Regulation.Temperature.SetPointAdjustment.Curve.Y1 := TO_REAL(Regulation.Temperature.Control.SP); 
	Regulation.Temperature.SetPointAdjustment.Curve.Y2 := TO_REAL(Regulation.Temperature.Control.SP); 
	Regulation.Temperature.SetPointAdjustment.Curve.Y3 := TO_REAL(Regulation.Temperature.Control.SP); 
	Regulation.Temperature.SetPointAdjustment.Curve.Y6 := TO_REAL(Regulation.Temperature.Control.SP); 
	Regulation.Temperature.SetPointAdjustment.Curve.Y7 := TO_REAL(Regulation.Temperature.Control.SP); 
	Regulation.Temperature.SetPointAdjustment.Curve.Y8 := TO_REAL(Regulation.Temperature.Control.SP); 
	Regulation.Temperature.SetPointAdjustment.Curve.Y9 := TO_REAL(Regulation.Temperature.Control.SP);
	Regulation.Temperature.Control.SP := 0;
	Regulation.SupplyAir.SetPointAdjustment.Curve.Y1 := TO_REAL(Regulation.SupplyAir.Control.SP);
	Regulation.SupplyAir.SetPointAdjustment.Curve.Y2 := TO_REAL(Regulation.SupplyAir.Control.SP);
	Regulation.SupplyAir.SetPointAdjustment.Curve.Y3 := TO_REAL(Regulation.SupplyAir.Control.SP);
	Regulation.SupplyAir.SetPointAdjustment.Curve.Y4 := TO_REAL(Regulation.SupplyAir.Control.SP);
	Regulation.SupplyAir.SetPointAdjustment.Curve.Y5 := TO_REAL(Regulation.SupplyAir.Control.SP);
	Regulation.SupplyAir.SetPointAdjustment.Curve.Y6 := TO_REAL(Regulation.SupplyAir.Control.SP);
	Regulation.SupplyAir.SetPointAdjustment.Curve.Y7 := TO_REAL(Regulation.SupplyAir.Control.SP);
	Regulation.SupplyAir.SetPointAdjustment.Curve.Y8 := TO_REAL(Regulation.SupplyAir.Control.SP);
	Regulation.SupplyAir.SetPointAdjustment.Curve.Y9 := TO_REAL(Regulation.SupplyAir.Control.SP);
	Regulation.SupplyAir.Control.SP := 0;
	Regulation.ExtractAir.SetPointAdjustment.Curve.Y1 := TO_REAL(Regulation.ExtractAir.Control.SP);
	Regulation.ExtractAir.SetPointAdjustment.Curve.Y2 := TO_REAL(Regulation.ExtractAir.Control.SP);
	Regulation.ExtractAir.SetPointAdjustment.Curve.Y3 := TO_REAL(Regulation.ExtractAir.Control.SP);
	Regulation.ExtractAir.SetPointAdjustment.Curve.Y4 := TO_REAL(Regulation.ExtractAir.Control.SP);
	Regulation.ExtractAir.SetPointAdjustment.Curve.Y5 := TO_REAL(Regulation.ExtractAir.Control.SP);
	Regulation.ExtractAir.SetPointAdjustment.Curve.Y6 := TO_REAL(Regulation.ExtractAir.Control.SP);
	Regulation.ExtractAir.SetPointAdjustment.Curve.Y7 := TO_REAL(Regulation.ExtractAir.Control.SP);
	Regulation.ExtractAir.SetPointAdjustment.Curve.Y8 := TO_REAL(Regulation.ExtractAir.Control.SP);
	Regulation.ExtractAir.SetPointAdjustment.Curve.Y9 := TO_REAL(Regulation.ExtractAir.Control.SP);
	Regulation.ExtractAir.Control.SP := 0;
	Regulation.LastApplyAbsoluteSetPointCurves := Regulation.ApplyAbsoluteSetPointCurves;
END_IF

NightCoolingHysteresis(Value := Parameters.IO.AIn.T_BT1, LimitValue := Parameters.Regulation.NightCoolingLimit, Offset := 0.5);
Parameters.Regulation.NightCooling := 
	Parameters.Regulation.NightCoolingRequest AND 
	NightCoolingHysteresis.Above AND 
	(NOT Parameters.System.Operation.TimeChannels.Q);
IF Parameters.Regulation.NightCoolingRequest AND NightCoolingHysteresis.Below THEN
	Parameters.Regulation.NightCoolingRequest := FALSE;
END_IF

END_FUNCTION_BLOCK

// ---- DUTs/Parameters/Regulation/AirParametersFB.TcPOU
FUNCTION_BLOCK AirParametersFB
VAR_IN_OUT
	Parameters: GreenMasterBaseParameters;
	ParametersFB: GreenMasterBaseParametersFB;
	AirParameters: AirParameters;
END_VAR
VAR_INPUT
END_VAR
VAR_OUTPUT
	SetPointAdjustmentFB: SetPointAdjustmentFB;
	TestOutput: LREAL := 3.14;
END_VAR
VAR
	LastControlMode: FanControlTypes;
END_VAR

IF AirParameters.ControlMode <> LastControlMode THEN
	CASE AirParameters.ControlMode OF
		FanControlTypes.Pressure:
			AirParameters.Control := AirParameters.Defaults.Pressure;
		FanControlTypes.Flow:
			AirParameters.Control := AirParameters.Defaults.Flow;
		FanControlTypes.Const:
			AirParameters.Control := AirParameters.Defaults.Const;
		FanControlTypes.SlaveFlow:
			AirParameters.Control := AirParameters.Defaults.SlaveFlow;
	END_CASE
	LastControlMode := AirParameters.ControlMode;
ELSIF Parameters.Regulation.SaveDefaults THEN
	CASE AirParameters.ControlMode OF
		FanControlTypes.Pressure:
			AirParameters.Defaults.Pressure := AirParameters.Control;
		FanControlTypes.Flow:
			AirParameters.Defaults.Flow := AirParameters.Control;
		FanControlTypes.Const:
			AirParameters.Defaults.Const := AirParameters.Control;
		FanControlTypes.SlaveFlow:
			AirParameters.Defaults.SlaveFlow := AirParameters.Control;
	END_CASE	
END_IF
SetPointAdjustmentFB(X := Parameters.Regulation.CompensationTemperature, SetPointAdjustment := AirParameters.SetPointAdjustment);
IF Parameters.IO.DIn.ExtendedOperation OR 
	(Parameters.System.Operation.TimeChannels.Q AND Parameters.System.Operation.TimeChannels.HighSpeed) OR
	(ADS_Standard.Tags.Settings.RemoteStart = 2) THEN
	AirParameters.Control.CSP := (AirParameters.Control.SP_HighSpeed + SetPointAdjustmentFB.Y) * AirParameters.AdjustCSP;
ELSE
	AirParameters.Control.CSP := (AirParameters.Control.SP + SetPointAdjustmentFB.Y) * AirParameters.AdjustCSP;
END_IF
IF AirParameters.Flow <> 0 THEN
	AirParameters.SpecificFanPower := AirParameters.Power / AirParameters.Flow;	
ELSE
	AirParameters.SpecificFanPower := 0;
END_IF
IF AirParameters.PressureRise <> 0 THEN
	AirParameters.FanEfficiency := AirParameters.SpecificFanPower / (AirParameters.PressureRise / 1000.0);
ELSE
	AirParameters.FanEfficiency := 0;
END_IF

END_FUNCTION_BLOCK

// ---- DUTs/Parameters/Regulation/SetPointAdjustmentFB.TcPOU
FUNCTION_BLOCK SetPointAdjustmentFB
VAR_IN_OUT
	SetPointAdjustment: SetPointAdjustment;
END_VAR
VAR_INPUT
	X: LREAL;
END_VAR
VAR_OUTPUT
	Y: LREAL;
END_VAR
VAR
	CurrentY: LREAL;
	LastY: LREAL;
END_VAR

CurrentY := 0;
LastY := SetPointAdjustment.Curve.Y1;
CurrentY := Interpolate(X := X, Y := CurrentY, X1 := SetPointAdjustment.Curve.X1, Y1 := SetPointAdjustment.Curve.Y1, X2 := SetPointAdjustment.Curve.X2, Y2 := SetPointAdjustment.Curve.Y2, LastY := LastY);
CurrentY := Interpolate(X := X, Y := CurrentY, X1 := SetPointAdjustment.Curve.X2, Y1 := SetPointAdjustment.Curve.Y2, X2 := SetPointAdjustment.Curve.X3, Y2 := SetPointAdjustment.Curve.Y3, LastY := LastY);
CurrentY := Interpolate(X := X, Y := CurrentY, X1 := SetPointAdjustment.Curve.X3, Y1 := SetPointAdjustment.Curve.Y3, X2 := SetPointAdjustment.Curve.X4, Y2 := SetPointAdjustment.Curve.Y4, LastY := LastY);
CurrentY := Interpolate(X := X, Y := CurrentY, X1 := SetPointAdjustment.Curve.X4, Y1 := SetPointAdjustment.Curve.Y4, X2 := SetPointAdjustment.Curve.X5, Y2 := SetPointAdjustment.Curve.Y5, LastY := LastY);
CurrentY := Interpolate(X := X, Y := CurrentY, X1 := SetPointAdjustment.Curve.X5, Y1 := SetPointAdjustment.Curve.Y5, X2 := SetPointAdjustment.Curve.X6, Y2 := SetPointAdjustment.Curve.Y6, LastY := LastY);
CurrentY := Interpolate(X := X, Y := CurrentY, X1 := SetPointAdjustment.Curve.X6, Y1 := SetPointAdjustment.Curve.Y6, X2 := SetPointAdjustment.Curve.X7, Y2 := SetPointAdjustment.Curve.Y7, LastY := LastY);
CurrentY := Interpolate(X := X, Y := CurrentY, X1 := SetPointAdjustment.Curve.X7, Y1 := SetPointAdjustment.Curve.Y7, X2 := SetPointAdjustment.Curve.X8, Y2 := SetPointAdjustment.Curve.Y8, LastY := LastY);
CurrentY := Interpolate(X := X, Y := CurrentY, X1 := SetPointAdjustment.Curve.X8, Y1 := SetPointAdjustment.Curve.Y8, X2 := SetPointAdjustment.Curve.X9, Y2 := SetPointAdjustment.Curve.Y9, LastY := LastY);
Y := CurrentY;
SetPointAdjustment.X := TO_REAL(X);
SetPointAdjustment.Y := TO_REAL(Y);

METHOD Interpolate : LREAL
VAR_IN_OUT
	LastY: LREAL;
END_VAR
VAR_INPUT
	X: LREAL;
	Y: LREAL;
	X1, Y1, X2, Y2: LREAL;
END_VAR
Interpolate := Y;
IF X2 > X1 THEN
	IF X > X2 THEN
		LastY := Y2;		
	END_IF
	IF (X >= X1) AND (X <= X2) THEN
		Interpolate := Y1 + ((X - X1) / (X2 - X1)) * (Y2 - Y1);
	ELSE
		Interpolate := LastY;
	END_IF
END_IF
END_METHOD

END_FUNCTION_BLOCK

// ---- DUTs/Controllers/Interpolate.TcPOU
FUNCTION_BLOCK Interpolate
VAR_INPUT
	EN: BOOL;
	x: LREAL;
END_VAR
VAR_OUTPUT
	ENO: BOOL;
	y: LREAL;
END_VAR
VAR CONSTANT
	NUM_POINTS: INT := 9;
END_VAR
VAR
	i: INT;
	j: INT;
	ss: LREAL;
	t: LREAL;
	k: LREAL;
END_VAR
VAR PERSISTENT
	xd: ARRAY [0..NUM_POINTS - 1] OF LREAL;
	yd: ARRAY [0..NUM_POINTS - 1] OF LREAL;
END_VAR

ENO := EN;
k := 0;
FOR i := 0 TO NUM_POINTS - 1 DO
	ss := 1;
	t := 1;
	FOR j := 0 TO NUM_POINTS - 1 DO
		IF i <> j THEN			
			ss := ss * (x - xd[j]);
			t := t * (xd[i] - xd[j]);
		END_IF
	END_FOR
	IF t <> 0 THEN
		k := k + ((ss / t) * yd[i]);		
	END_IF
END_FOR
y := k;

END_FUNCTION_BLOCK

// ---- DUTs/Fans/SpecificFanPower.TcPOU
FUNCTION_BLOCK SpecificFanPower
VAR_INPUT
END_VAR
VAR_OUTPUT
END_VAR
VAR
END_VAR

END_FUNCTION_BLOCK

// ---- DUTs/Parameters/Regulation/TemperatureControlParametersFB.TcPOU
FUNCTION_BLOCK TemperatureControlParametersFB
VAR_IN_OUT
	Parameters: GreenMasterBaseParameters;
	ParametersFB: GreenMasterBaseParametersFB;
	Temperature: TemperatureControlParameters;
END_VAR
VAR_INPUT
END_VAR
VAR_OUTPUT
	SetPointAdjustmentFB: SetPointAdjustmentFB;
END_VAR
VAR
END_VAR

SetPointAdjustmentFB(X := Parameters.Regulation.CompensationTemperature, SetPointAdjustment := Parameters.Regulation.Temperature.SetPointAdjustment);
Parameters.Regulation.Temperature.Control.CSP := MAX(Parameters.Regulation.Temperature.Control.SP + Temperature.SetPointAdjustment.Y, 4);
IF Parameters.Regulation.NightCooling THEN
	Parameters.Regulation.Temperature.Control.CSP := Parameters.Regulation.NightCoolingLimit;
END_IF
IF (Main.GreenMaster.GetState() = SystemStates.Run) AND (Main.GreenMaster.StateTime() > LTIME#1M) THEN
	Parameters.Regulation.Temperature.Efficiency := CalculateEfficiency(Parameters.IO.AIn.T_BT3, Parameters.IO.AIn.T_BT2, Parameters.IO.AIn.F_BT1);
	IF ((Parameters.IO.AOut.F_QN1 < 0.001) AND (Parameters.Regulation.Temperature.HeaterOutputDirection = HeaterOutputDirections.DecreaseToHeat)) OR
		((Parameters.IO.AOut.F_QN1 > 0.999) AND (Parameters.Regulation.Temperature.HeaterOutputDirection = HeaterOutputDirections.IncreaseToHeat)) THEN
		Parameters.Alarm.Status.B.HeatExchangerEfficiency := Parameters.Regulation.Temperature.Efficiency < Parameters.Alarm.Limits.B.HeatExchangerEfficiency;
	ELSE
		Parameters.Alarm.Status.B.HeatExchangerEfficiency := FALSE;
	END_IF
ELSE
	Parameters.Regulation.Temperature.Efficiency := 0;	
	Parameters.Alarm.Status.B.HeatExchangerEfficiency := FALSE;
END_IF

METHOD MaxOutput : LREAL
VAR_INPUT
END_VAR
IF Temperature.HeaterOutputDirection = HeaterOutputDirections.IncreaseToHeat THEN
	MaxOutput := 1;
ELSE
	MaxOutput := 0;
END_IF
END_METHOD

METHOD MinOutput : LREAL
VAR_INPUT
END_VAR
IF Temperature.HeaterOutputDirection = HeaterOutputDirections.IncreaseToHeat THEN
	MinOutput := 0;
ELSE
	MinOutput := 1;
END_IF
END_METHOD

END_FUNCTION_BLOCK

// ---- DUTs/Utilities/CalculateEfficiency.TcPOU
FUNCTION CalculateEfficiency : lreal
VAR_INPUT
	T_BT3: LREAL;
	T_BT2: LREAL;
	F_BT1: LREAL;
END_VAR
VAR
	denom: LREAL;
END_VAR

(*
Verkningsgradsberäkning + verkningsgradslarm

(T.BT3-T.BT2) / (F.BT1-T.BT2)

Just nu (i fabriken finns aldrig optimala förhållanden då de omgivande temperaturerna är ganska lika):
(20,7-20,5) / (21,0-20,5) = 0,4 = 40% verkningsgrad

Exempel på en norm-installation:
(21-10) / (22-10) = 0,9166 = 91,7% verkningsgrad


PRESENTATION AV VERKNINGSGRAD
-----------------------------
OBS! Presentation av verkningsgrad får ALDRIG överstiga 100%, även om beräkningen säger att det kan bli så. Det kan hända vid okalibrerade givare eller vid ovanliga omgivande temperaturer. 

Exempel på högre verkningsgrad än 100%:
Om tilluften är 21 grader och utetemperaturen är 20 grader
samtidigt som frånluften är 20,5 grader så kommer beräkningen visa 200% verkningsgrad

(21-20) / (20,5-20) = 2

Sådana här fall uppkommer väldigt sällan, men vi har stött på det under vissa förhållanden i tidigare system, så det är otroligt viktigt att OM verkningsgradsberäkningen visar över 100% så skall det presenterade värdet vara 100%, ALDRIG högre! Jag har aldrig stött på att man kan få ett negativt resultat, men samma försäkran borde ändå läggas in åt andra hållet, verkningsgraden kan ju aldrig bli lägre än 0%. (Skalan på verkningsgrad är alltså uteslutande 0-100%) 


VERKNINGSGRADSLARM
------------------------------------------
Om värmeväxlaren ligger i full återvinning (0% öppet F.QN1 för fallet med GMXXL) och verkningsgraden understiger XX % under YY sekunder sätts verkningsgradslarm. Verkningsgradslarmet "maskas" om värmeåtervinningen ligger i kylläge, dvs. så fort F.QN1 är över 0%, då skall man aldrig erhålla verkningsgradslarm. (Tex vår och sommar)

*)
denom := F_BT1-T_BT2;
IF denom > 0 THEN
	CalculateEfficiency := (T_BT3-T_BT2) / (F_BT1-T_BT2);
	IF CalculateEfficiency > 1 THEN
		CalculateEfficiency := 1;
	END_IF
	IF CalculateEfficiency < 0 THEN
		CalculateEfficiency := 0;
	END_IF
ELSE
	CalculateEfficiency := 1;
END_IF

END_FUNCTION

// ---- DUTs/Utilities/Hysteresis.TcPOU
FUNCTION_BLOCK Hysteresis
VAR_INPUT
	EN: BOOL := TRUE;
	Value: LREAL;
	LimitValue: LREAL;
	Offset: LREAL; 
END_VAR
VAR_OUTPUT
	ENO: BOOL;
	Above: BOOL;
	Below: BOOL;
END_VAR
VAR
	Hysteresis: INT;
	CurValue: LREAL;
	PreValue: LREAL;
	HystLimit: LREAL;
	HystOffset: LREAL;
END_VAR

HystLimit := LimitValue;
HystOffset := Offset;
IF EN THEN
	Update(Value);
ELSE
	Reset();
END_IF
PreValue := CurValue;
CurValue := Value;
ENO := EN;

METHOD Reset
VAR_INPUT
END_VAR
Hysteresis := 0;
Above := FALSE;
Below := FALSE;
END_METHOD

METHOD PRIVATE Update
VAR_INPUT
	Value: LREAL; 
END_VAR
IF ABS(Value - HystLimit) >= ABS(HystOffset) THEN
	Hysteresis := 0;
END_IF
IF (Value > (LimitValue + Offset * Hysteresis)) AND (PreValue <= (LimitValue + Offset * Hysteresis)) THEN
	IF Hysteresis > -1 THEN
		Hysteresis := Hysteresis - 1;
	END_IF
END_IF
IF (Value <= (LimitValue + Offset * Hysteresis)) AND (PreValue > (LimitValue + Offset * Hysteresis)) THEN
	IF Hysteresis < 1 THEN
		Hysteresis := Hysteresis + 1;
	END_IF
END_IF
Above := CurValue > (LimitValue + HystOffset * Hysteresis);
Below := CurValue <= (LimitValue + HystOffset * Hysteresis);
END_METHOD

END_FUNCTION_BLOCK

// ---- DUTs/Utilities/LimitValue.TcPOU
FUNCTION LimitValue : LREAL
VAR_INPUT
	Value: LREAL;
	MinValue: LREAL;
	MaxValue: LREAL;
END_VAR
VAR
  Res: LREAL;
END_VAR

Res := Value;
IF Res < MinValue THEN
	Res := MinValue;
END_IF;
IF Res > MaxValue THEN
	Res := MaxValue;
END_IF;
LimitValue := Res;

END_FUNCTION

// ---- DUTs/Parameters/IO/IOParametersFB.TcPOU
FUNCTION_BLOCK IOParametersFB
VAR_IN_OUT
	GreenMaster: GreenMasterBase;
	Parameters: GreenMasterBaseParameters;
	ParametersFB: GreenMasterBaseParametersFB;
END_VAR
VAR_INPUT
END_VAR
VAR_OUTPUT
	DIn: DigitalInputParametersFB;
	//DInLevels: DigitalInputLevelsFB;
	DOut: DigitalOutputParametersFB;
	//DOutOverride: DigitalOutputOverrideParametersFB;
	AIn: AnalogInputParametersFB;
	AOut: AnalogOutputParametersFB;
	//AOutOverride: AnalogOutputOverrideParametersFB;
	//AOutCalibration: AnalogOutputCalibrationFB;
	//Status: IoStatusFB;
END_VAR
VAR
	AnySensorError: BOOL;
	StartTime: Timer;
END_VAR

Parameters.IO.Status.InputStatus.AI01 := BoolToErrorText(Globals.IO.AIn.AI01_Error); 
Parameters.IO.Status.InputStatus.AI02 := BoolToErrorText(Globals.IO.AIn.AI02_Error); 
Parameters.IO.Status.InputStatus.AI03 := BoolToErrorText(Globals.IO.AIn.AI03_Error); 
Parameters.IO.Status.InputStatus.AI04 := BoolToErrorText(Globals.IO.AIn.AI04_Error); 
Parameters.IO.Status.InputStatus.AI05 := BoolToErrorText(Globals.IO.AIn.AI05_Error); 
Parameters.IO.Status.InputStatus.AI06 := BoolToErrorText(Globals.IO.AIn.AI06_Error); 
Parameters.IO.Status.InputStatus.AI07 := BoolToErrorText(Globals.IO.AIn.AI07_Error); 
Parameters.IO.Status.InputStatus.AI08 := BoolToErrorText(Globals.IO.AIn.AI08_Error); 
Parameters.IO.Status.InputStatus.AI09 := BoolToErrorText(Globals.IO.AIn.AI09_Error); 
Parameters.IO.Status.InputStatus.AI10 := BoolToErrorText(Globals.IO.AIn.AI10_Error); 
Parameters.IO.Status.InputStatus.AI11 := BoolToErrorText(Globals.IO.AIn.AI11_Error); 
Parameters.IO.Status.InputStatus.AI12 := BoolToErrorText(Globals.IO.AIn.AI12_Error); 
Parameters.IO.Status.InputStatus.AI13 := BoolToErrorText(Globals.IO.AIn.AI13_Error);
Parameters.IO.Status.InputStatus.AI14 := BoolToErrorText(Globals.IO.AIn.AI14_Error); 
Parameters.IO.Status.InputStatus.AI15 := BoolToErrorText(Globals.IO.AIn.AI15_Error); 
Parameters.IO.Status.InputStatus.AI16 := BoolToErrorText(Globals.IO.AIn.AI16_Error); 
Parameters.IO.Status.InputStatus.AI17 := BoolToErrorText(Globals.IO.AIn.AI17_Error); 
Parameters.IO.Status.InputStatus.AI18 := BoolToErrorText(Globals.IO.AIn.AI18_Error); 
Parameters.IO.Status.InputStatus.AI19 := BoolToErrorText(Globals.IO.AIn.AI19_Error); 
Parameters.IO.Status.InputStatus.AI20 := BoolToErrorText(Globals.IO.AIn.AI20_Error); 
Parameters.IO.Status.InputStatus.AI21 := BoolToErrorText(Globals.IO.AIn.AI21_Error); 
Parameters.IO.Status.InputStatus.AI22 := BoolToErrorText(Globals.IO.AIn.AI22_Error); 
Parameters.IO.Status.InputStatus.AI23 := BoolToErrorText(Globals.IO.AIn.AI23_Error); 
Parameters.IO.Status.InputStatus.AI24 := BoolToErrorText(Globals.IO.AIn.AI24_Error); 

Parameters.IO.Status.SensorStatus.F_BT1 := BoolToErrorText(Globals.IO.AIn.AI01_Error); 
Parameters.IO.Status.SensorStatus.T_BT2 := BoolToErrorText(Globals.IO.AIn.AI02_Error);
Parameters.IO.Status.SensorStatus.T_BT3 := BoolToErrorText(Globals.IO.AIn.AI03_Error);
Parameters.IO.Status.SensorStatus.H_BT1 := BoolToErrorText(Globals.IO.AIn.AI04_Error);
Parameters.IO.Status.SensorStatus.T_BT1 := BoolToErrorText(Globals.IO.AIn.AI05_Error); 
Parameters.IO.Status.SensorStatus.BT1 := BoolToErrorText(Globals.IO.AIn.AI06_Error);
Parameters.IO.Status.SensorStatus.BT2 := BoolToErrorText(Globals.IO.AIn.AI07_Error);
Parameters.IO.Status.SensorStatus.F_BT2 := BoolToErrorText(Globals.IO.AIn.AI08_Error);

IF NOT Main.UseKL3464 THEN
	Parameters.IO.Status.SensorStatus.F_BP1 := BoolToErrorText(GreenMaster.AI2.F_BP1_Error);
	Parameters.IO.Status.SensorStatus.T_BP1 := BoolToErrorText(GreenMaster.AI2.T_BP1_Error);
ELSE
	Parameters.IO.Status.SensorStatus.F_BP1 := BoolToErrorText(Globals.AI3468.AI2_Error);
	Parameters.IO.Status.SensorStatus.T_BP1 := BoolToErrorText(Globals.AI3468.AI1_Error);
END_IF
Parameters.IO.Status.SensorStatus.F_BP2 := BoolToErrorText(GreenMaster.AI2.F_BP2_Error);
Parameters.IO.Status.SensorStatus.T_BP2 := BoolToErrorText(GreenMaster.AI2.T_BP2_Error);
Parameters.IO.Status.SensorStatus.F_BP3 := BoolToErrorText(GreenMaster.AI2.F_BP3_Error);
Parameters.IO.Status.SensorStatus.T_BF1 := BoolToErrorText(GreenMaster.AI2.T_BF1_Error);
Parameters.IO.Status.SensorStatus.F_BF1 := BoolToErrorText(GreenMaster.AI2.F_BF1_Error);	

StartTime();
IF (StartTime.ET > LTIME#20S) and (not Parameters.System.Operation.Simulation) THEN
	// Check if any sensor error
	AnySensorError := FALSE;
	AnySensorError := AnySensorError OR Globals.IO.AIn.AI01_Error; 
	AnySensorError := AnySensorError OR Globals.IO.AIn.AI02_Error;
	AnySensorError := AnySensorError OR Globals.IO.AIn.AI03_Error;
	AnySensorError := AnySensorError OR Globals.IO.AIn.AI04_Error;
	AnySensorError := AnySensorError OR Globals.IO.AIn.AI05_Error; 
	AnySensorError := AnySensorError OR Globals.IO.AIn.AI06_Error;
	AnySensorError := AnySensorError OR Globals.IO.AIn.AI07_Error;
	AnySensorError := AnySensorError OR Globals.IO.AIn.AI08_Error;
	
	AnySensorError := AnySensorError OR GreenMaster.AI2.F_BP1_Error;
	AnySensorError := AnySensorError OR GreenMaster.AI2.T_BP1_Error;
	AnySensorError := AnySensorError OR GreenMaster.AI2.F_BP2_Error;
	AnySensorError := AnySensorError OR GreenMaster.AI2.T_BP2_Error;
	AnySensorError := AnySensorError OR GreenMaster.AI2.F_BP3_Error;
	AnySensorError := AnySensorError OR GreenMaster.AI2.T_BF1_Error;
	AnySensorError := AnySensorError OR GreenMaster.AI2.F_BF1_Error;	
	
END_IF

END_FUNCTION_BLOCK

// ---- DUTs/Parameters/IO/DigitalInputParametersFB.TcPOU
FUNCTION_BLOCK DigitalInputParametersFB
VAR_INPUT
END_VAR
VAR_OUTPUT
END_VAR
VAR
END_VAR

METHOD Update : BOOL
VAR_INPUT
	DI: REFERENCE TO GreenMasterDI_Base;
	Parameters: REFERENCE TO GreenMasterBaseParameters;
	DIn: reference to DigitalInputParameters;
END_VAR
IF NOT Parameters.System.Operation.Simulation THEN
	DIn.AUTO := DI.AUTO;
	DIn.FireExtractAlarm := DI.FireExtractAlarm;
	DIn.FuseAlarm := DI.FuseAlarm;
	DIn.HAND := DI.Hand;
	DIn.T_GQ1_Alarm := DI.T_GQ1_Alarm;
	DIn.F_GQ1_Alarm := DI.F_GQ1_Alarm;
	DIn.F_QM2_Closed := DI.F_QM2_Closed;
	DIn.F_QM2_Open := DI.F_QM2_Open;
	DIn.ExtendedOperation := DI.ExtendedOperation;
	DIn.ServiceAlarmCentralAndSmokeExhaustAir := DI.ServiceAlarmCentralAndSmokeExhaustAir;
	DIn.FireSupplyAlarm := DI.FireSupplyAlarm;
	DIn.ServiceAlarmSupplyAir := DI.ServiceAlarmSupplyAir;
	DIn.H_GP1_Running := DI.H_GP1_Running;
	DIn.H_GP1_Alarm := DI.H_GP1_Alarm;
	DIn.C_GP1_Running := DI.C_GP1_Running;
	DIn.C_GP1_Alarm := DI.C_GP1_Alarm;
	DIn.TX1_Running := DI.TX1_Running;
	DIn.ResetAlarm := DI.ResetAlarm;
	DIn.P2_Running := DI.P2_Running;
	DIn.ExpansionVesselAlarm := DI.ExpansionVesselAlarm;
	DIn.FirePanelSupplyStart := DI.FireActivateSupplyAir;
	DIn.FirePanelSupplyStop := DI.FireDeactivateSupplyAir;
	DIn.FirePanelExtractStart := DI.FireActivateExtractAir;
	DIn.FirePanelExtractStop := DI.FireDeactivateExtractAir;
END_IF
END_METHOD

END_FUNCTION_BLOCK

// ---- DUTs/GreenMaster/IO/GreenMasterDI_Base.TcPOU
FUNCTION_BLOCK GreenMasterDI_Base
VAR_IN_OUT
	DIn: DigitalInputs;
	DInLevels: DigitalInputLevels;
END_VAR
VAR_INPUT
END_VAR
VAR_OUTPUT
	Auto: BOOL;
	FireExtractAlarm: BOOL;
	FuseAlarm: BOOL;
	Hand: BOOL;
	T_GQ1_Alarm: BOOL;
	F_GQ1_Alarm: BOOL;
	T_QM2_Closed: BOOL;
	T_QM2_Open: BOOL;
	F_QM1_Closed: BOOL;
	F_QM1_Open: BOOL;
	F_QM2_Closed: BOOL;
	F_QM2_Open: BOOL;
	ExtendedOperation: BOOL;
	ServiceAlarmCentralAndSmokeExhaustAir: BOOL;
	FireSupplyAlarm: BOOL;
	ServiceAlarmSupplyAir: BOOL;
	H_GP1_Running: BOOL;
	C_GP1_Running: BOOL;
	H_GP1_Alarm: BOOL;
	C_GP1_Alarm: BOOL;
	TX1_Running: BOOL;
	ResetAlarm: BOOL;
	P2_Running: BOOL;
	P2_Alarm: BOOL;
	ExpansionVesselAlarm: BOOL;
	FireActivateSupplyAir: BOOL;
	FireDeactivateSupplyAir: BOOL;
	FireActivateExtractAir: BOOL;
	FireDeactivateExtractAir: BOOL;
END_VAR
VAR
END_VAR

END_FUNCTION_BLOCK

// ---- DUTs/Parameters/IO/DigitalOutputParametersFB.TcPOU
FUNCTION_BLOCK DigitalOutputParametersFB
VAR_INPUT
	DOut: DigitalOutputParameters;
END_VAR
VAR_OUTPUT
	H_GP1_OnTime: LTIME;
	F_QM1_OnTime: LTIME;
	F_QM2_OnTime: LTIME;
	T_QM2_OnTime: LTIME;
END_VAR
VAR
	H_GP1_LTON: Timer; // $(skip)
	F_QM1_LTON: Timer; // $(skip)
	F_QM2_LTON: Timer; // $(skip)
	T_QM2_LTON: Timer; // $(skip)
END_VAR

H_GP1_LTON(EN := DOut.H_GP1, ET => H_GP1_OnTime);
F_QM1_LTON(EN := DOut.F_QM1, ET => F_QM1_OnTime);
F_QM2_LTON(EN := DOut.F_QM2, ET => F_QM2_OnTime);
T_QM2_LTON(EN := DOut.T_QM2, ET => T_QM2_OnTime);

METHOD Update : BOOL
VAR_INPUT
	DO_: REFERENCE TO GreenMasterDO_Base;
	Parameters: REFERENCE TO GreenMasterBaseParameters;
	EnableWriteDampers: BOOL := TRUE;
END_VAR
VAR
	NotFire: BOOL;
END_VAR
NotFire := NOT Main.GreenMaster.FireAlarm();
DO_.H_GP1 := ifc_bool(Parameters.IO.DOutOverride.H_GP1_Override AND NotFire, Parameters.IO.DOutOverride.H_GP1_OverrideValue, Parameters.IO.DOut.H_GP1);
DO_.C_GP1 := ifc_bool(Parameters.IO.DOutOverride.C_GP1_Override AND NotFire, Parameters.IO.DOutOverride.C_GP1_OverrideValue, Parameters.IO.DOut.C_GP1);
IF EnableWriteDampers THEN
	DO_.F_QM1 := ifc_bool(Parameters.IO.DOutOverride.F_QM1_Override AND NotFire, Parameters.IO.DOutOverride.F_QM1_OverrideValue, Parameters.IO.DOut.F_QM1);
	DO_.T_QM2 := ifc_bool(Parameters.IO.DOutOverride.T_QM2_Override AND NotFire, Parameters.IO.DOutOverride.T_QM2_OverrideValue, Parameters.IO.DOut.T_QM2);
END_IF
DO_.R_QM1 := ifc_bool(Parameters.IO.DOutOverride.R_QM1_Override AND NotFire, Parameters.IO.DOutOverride.R_QM1_OverrideValue, Parameters.IO.DOut.R_QM1);
DO_.F_QM2 := ifc_bool(Parameters.IO.DOutOverride.F_QM2_Override AND NotFire, Parameters.IO.DOutOverride.F_QM2_OverrideValue, Parameters.IO.DOut.F_QM2);
DO_.T_QM1_1 := ifc_bool(Parameters.IO.DOutOverride.T_QM1_1_Override AND NotFire, Parameters.IO.DOutOverride.T_QM1_1_OverrideValue, Parameters.IO.DOut.T_QM1_1);
DO_.T_QM1_2 := ifc_bool(Parameters.IO.DOutOverride.T_QM1_2_Override AND NotFire, Parameters.IO.DOutOverride.T_QM1_2_OverrideValue, Parameters.IO.DOut.T_QM1_2);
DO_.T_QM1_3 := ifc_bool(Parameters.IO.DOutOverride.T_QM1_3_Override AND NotFire, Parameters.IO.DOutOverride.T_QM1_3_OverrideValue, Parameters.IO.DOut.T_QM1_3);
DO_.T_QM1_4 := ifc_bool(Parameters.IO.DOutOverride.T_QM1_4_Override AND NotFire, Parameters.IO.DOutOverride.T_QM1_4_OverrideValue, Parameters.IO.DOut.T_QM1_4);
DO_.T_QM1_5 := ifc_bool(Parameters.IO.DOutOverride.T_QM1_5_Override AND NotFire, Parameters.IO.DOutOverride.T_QM1_5_OverrideValue, Parameters.IO.DOut.T_QM1_5);
DO_.T_QM1_6 := ifc_bool(Parameters.IO.DOutOverride.T_QM1_6_Override AND NotFire, Parameters.IO.DOutOverride.T_QM1_6_OverrideValue, Parameters.IO.DOut.T_QM1_6);
Parameters.IO.DOut.F_QM2_ActiveWhenStopped := FALSE;
DO_.SupplyRunning := Parameters.IO.DOut.T_RUN;
DO_.ExhaustRunning := Parameters.IO.DOut.F_RUN;

DO_.AlarmRelayA := Parameters.IO.DOut.AL_A;
DO_.AlarmRelayB := Parameters.IO.DOut.AL_B;
DO_.AlarmRelayC := Parameters.IO.DOut.AL_C;
DO_.AlarmRelayD := Parameters.IO.DOut.AL_D;
END_METHOD

END_FUNCTION_BLOCK

// ---- DUTs/Utilities/Timer.TcPOU
FUNCTION_BLOCK Timer
VAR_INPUT
	EN: BOOL := TRUE;
END_VAR
VAR_OUTPUT
	ET: LTIME;
END_VAR
VAR
    _TimeTick: LINT;
    _StartTick: LINT;
    _Timeout: BOOL;
END_VAR

ET := LINT_TO_LTIME(ElapsedTime() * 1000000);
IF NOT EN THEN
	Restart();
END_IF

METHOD ElapsedTime : LINT
VAR_INPUT
END_VAR
IF EN THEN
	ElapsedTime := (GetTickCount() - _StartTick);
ELSE
	ElapsedTime := 0;	
END_IF
END_METHOD

METHOD FB_init : BOOL
VAR_INPUT
	bInitRetains : BOOL; // if TRUE, the retain variables are initialized (warm start / cold start)
	bInCopyCode : BOOL;  // if TRUE, the instance afterwards gets moved into the copy code (online change)
END_VAR
TimeoutTime := 1000;
Restart();
END_METHOD

METHOD Restart : BOOL
VAR_INPUT
END_VAR
_Timeout := FALSE;
_StartTick := GetTickCount();
Restart := TRUE;
END_METHOD

METHOD Timeout : BOOL
VAR_INPUT
END_VAR
IF NOT _Timeout THEN
	IF (GetTickCount() - _StartTick) >= _TimeTick THEN
		_Timeout := TRUE;
	END_IF
END_IF
Timeout := _Timeout;
END_METHOD

PROPERTY TimeoutTime : LINT
GET
TimeoutTime := _TimeTick;
END_GET
SET
VAR
	Temp: lint;
END_VAR
Temp := TimeoutTime;
IF (TimeoutTime > 0) AND (Temp <= 1) THEN
	Temp := 2; { Smallest timeout }
END_IF
IF Temp <> _TimeTick THEN
	_TimeTick := Temp;
	Restart();
END_IF
END_SET
END_PROPERTY

END_FUNCTION_BLOCK

// ---- DUTs/Utilities/GetTickCount.TcPOU
FUNCTION GetTickCount : LINT
VAR_INPUT
END_VAR
VAR
	
END_VAR
VAR_STAT
	GST: Tc2_System.GETCPUCOUNTER;
END_VAR

GST();
GetTickCount := LWORD_TO_LINT(((DWORD_TO_LWORD(GST.cpuCntHiDW) * 16#100000000) + GST.cpuCntLoDW)) / 10000;

END_FUNCTION

// ---- DUTs/GreenMaster/IO/GreenMasterDO_Base.TcPOU
FUNCTION_BLOCK GreenMasterDO_Base
VAR_IN_OUT
	DOut: DigitalOutputs;
END_VAR
VAR_INPUT
	H_GP1: BOOL;
	C_GP1: BOOL;
	ExhaustRunning: BOOL;
	F_QM1: BOOL;
	T_QM2: BOOL;
	R_QM1: BOOL;
	F_QM2: BOOL;
	SupplyRunning: BOOL;
	T_QM1_1: BOOL;
	T_QM1_2: BOOL;
	T_QM1_3: BOOL;
	T_QM1_4: BOOL;
	T_QM1_5: BOOL;
	T_QM1_6: BOOL;			
	AlarmRelayA: BOOL;
	AlarmRelayB: BOOL;
	AlarmRelayC: BOOL;
	AlarmRelayD: BOOL;
	P2: BOOL;
END_VAR
VAR_OUTPUT
END_VAR
VAR
END_VAR

END_FUNCTION_BLOCK

// ---- DUTs/Utilities/ifc_bool.TcPOU
FUNCTION ifc_bool : BOOL
VAR_INPUT
	Condition: BOOL;
	ValueTrue: BOOL;
	ValueFalse: BOOL;
END_VAR
VAR
END_VAR

IF Condition THEN
	ifc_bool := ValueTrue;
ELSE
	ifc_bool := ValueFalse;
END_IF

END_FUNCTION

// ---- DUTs/Parameters/IO/AnalogInputParametersFB.TcPOU
FUNCTION_BLOCK AnalogInputParametersFB
VAR_INPUT
END_VAR
VAR_OUTPUT
END_VAR
VAR
END_VAR

METHOD Update : BOOL
VAR_INPUT
	AI: REFERENCE TO GreenMasterAI_Base;
	AI2: REFERENCE TO GreenMasterAIU_Base;
	Parameters: REFERENCE TO GreenMasterBaseParameters;
END_VAR

VAR
END_VAR
IF NOT Parameters.System.Operation.Simulation THEN
	Parameters.IO.AIn.F_BT1 := AI.F_BT1;
	Parameters.IO.AIn.F_BT1_Error := AI.F_BT1_Error AND Parameters.IO.AIn.F_BT1_EN;
	Parameters.IO.AIn.T_BT2 := AI.T_BT2;
	Parameters.IO.AIn.T_BT2_Error := AI.T_BT2_Error AND Parameters.IO.AIn.T_BT2_EN;
	Parameters.IO.AIn.T_BT3 := AI.T_BT3;
	Parameters.IO.AIn.T_BT3_Error := AI.T_BT3_Error AND Parameters.IO.AIn.T_BT3_EN;
	Parameters.IO.AIn.H_BT1 := AI.H_BT1;
	Parameters.IO.AIn.H_BT1_Error := AI.H_BT1_Error AND Parameters.IO.AIn.H_BT1_EN;
	Parameters.IO.AIn.T_BT1 := AI.T_BT1; 
	Parameters.IO.AIn.T_BT1_Error := AI.T_BT1_Error AND Parameters.IO.AIn.T_BT1_EN;
	Parameters.IO.AIn.BT1 := AI.BT1;
	Parameters.IO.AIn.BT1_Error := AI.BT1_Error AND Parameters.IO.AIn.BT1_EN;
	Parameters.IO.AIn.BT2 := AI.BT2;
	Parameters.IO.AIn.BT2_Error := AI.BT2_Error AND Parameters.IO.AIn.BT2_EN;
	Parameters.IO.AIn.F_BT2 := AI.F_BT2;
	Parameters.IO.AIn.F_BT2_Error := AI.F_BT2_Error AND Parameters.IO.AIn.F_BT2_EN;
	IF Main.UseKL3464 THEN
		Parameters.IO.AIn.T_BP1 := 500 * (TO_LREAL(Globals.AI3468.AI1) / 32767.0);
		Parameters.IO.AIn.T_BP1_Error := Globals.AI3468.AI2_Error;
		Parameters.IO.AIn.F_BP1 := 500 * (TO_LREAL(Globals.AI3468.AI2) / 32767.0);
		Parameters.IO.AIn.F_BP1_Error := Globals.AI3468.AI1_Error;
	ELSE
		Parameters.IO.AIn.F_BP1 := AI2.F_BP1;
		Parameters.IO.AIn.F_BP1_Error := AI2.F_BP1_Error AND Parameters.IO.AIn.F_BP1_EN;
		Parameters.IO.AIn.T_BP1 := AI2.T_BP1;
		Parameters.IO.AIn.T_BP1_Error := AI2.T_BP1_Error AND Parameters.IO.AIn.T_BP1_EN;
	END_IF
	Parameters.IO.AIn.F_BP2 := AI2.F_BP2;
	Parameters.IO.AIn.F_BP2_Error := AI2.F_BP2_Error AND Parameters.IO.AIn.F_BP2_EN;
	Parameters.IO.AIn.T_BP2 := AI2.T_BP2;
	Parameters.IO.AIn.T_BP2_Error := AI2.T_BP2_Error AND Parameters.IO.AIn.T_BP2_EN;
	Parameters.IO.AIn.F_BP3 := AI2.F_BP3;
	Parameters.IO.AIn.F_BP3_Error := AI2.F_BP3_Error AND Parameters.IO.AIn.F_BP3_EN;
	Parameters.IO.AIn.T_BF1 := AI2.T_BF1;
	Parameters.IO.AIn.T_BF1_Error := AI2.T_BF1_Error AND Parameters.IO.AIn.T_BF1_EN;
	Parameters.IO.AIn.F_BF1 := AI2.F_BF1;	
	Parameters.IO.AIn.F_BF1_Error := AI2.F_BF1_Error AND Parameters.IO.AIn.F_BF1_EN;
ELSE
	(*
	Parameters.IO.AIn.F_BT1_Error := FALSE;
	Parameters.IO.AIn.T_BT2_Error := FALSE;
	Parameters.IO.AIn.T_BT3_Error := FALSE;
	Parameters.IO.AIn.H_BT1_Error := FALSE;
	Parameters.IO.AIn.T_BT1_Error := FALSE;
	Parameters.IO.AIn.BT1_Error := FALSE;
	Parameters.IO.AIn.BT2_Error := FALSE;
	Parameters.IO.AIn.F_BT2_Error := FALSE;
	Parameters.IO.AIn.F_BP1_Error := FALSE;
	Parameters.IO.AIn.T_BP1_Error := FALSE;
	Parameters.IO.AIn.F_BP2_Error := FALSE;
	Parameters.IO.AIn.T_BP2_Error := FALSE;
	Parameters.IO.AIn.F_BP3_Error := FALSE;
	Parameters.IO.AIn.T_BF1_Error := FALSE;
	Parameters.IO.AIn.F_BF1_Error := FALSE;
	*)
END_IF
END_METHOD

END_FUNCTION_BLOCK

